LIN {X -0.030,Y -571.399,Z 1067.188,A 0.000,B 0.000,C 90.000,E1 69.752} C_DIS
LIN {X -0.071,Y -572.958,Z 1067.177,A 0.000,B 0.000,C 90.000,E1 67.847} C_DIS
LIN {X -0.064,Y -573.976,Z 1067.169,A 0.000,B 0.000,C 90.000,E1 66.485} C_DIS
LIN {X -0.020,Y -574.631,Z 1067.165,A 0.000,B 0.000,C 90.000,E1 65.665} C_DIS
LIN {X 0.089,Y -575.617,Z 1067.156,A 0.000,B 0.000,C 90.000,E1 64.024} C_DIS
LIN {X -0.046,Y -576.546,Z 1067.147,A 0.000,B 0.000,C 90.000,E1 62.410} C_DIS
LIN {X -0.162,Y -577.447,Z 1067.138,A 0.000,B 0.000,C 90.000,E1 60.795} C_DIS
LIN {X 0.161,Y -578.076,Z 1067.130,A 0.000,B 0.000,C 90.000,E1 59.410} C_DIS
LIN {X 0.146,Y -578.736,Z 1067.121,A 0.000,B 0.000,C 90.000,E1 57.788} C_DIS
LIN {X 0.303,Y -579.331,Z 1067.114,A 0.000,B 0.000,C 90.000,E1 56.421} C_DIS
LIN {X 0.155,Y -579.956,Z 1067.105,A 0.000,B 0.000,C 90.000,E1 54.815} C_DIS
LIN {X 0.019,Y -580.235,Z 1067.099,A 0.000,B 0.000,C 90.000,E1 53.749} C_DIS
LIN {X 0.058,Y -580.388,Z 1067.091,A 0.000,B 0.000,C 90.000,E1 52.396} C_DIS
LIN {X -0.248,Y -580.373,Z 1067.087,A 0.000,B 0.000,C 90.000,E1 51.618} C_DIS
LIN {X -0.198,Y -580.244,Z 1067.082,A 0.000,B 0.000,C 90.000,E1 50.803} C_DIS
LIN {X -0.386,Y -579.481,Z 1067.072,A 0.000,B 0.000,C 90.000,E1 48.933} C_DIS
LIN {X -0.089,Y -578.838,Z 1067.064,A 0.000,B 0.000,C 90.000,E1 47.553} C_DIS
LIN {X 0.044,Y -578.138,Z 1067.058,A 0.000,B 0.000,C 90.000,E1 46.458} C_DIS
LIN {X -0.249,Y -577.299,Z 1067.052,A 0.000,B 0.000,C 90.000,E1 45.405} C_DIS
LIN {X -0.269,Y -576.458,Z 1067.048,A 0.000,B 0.000,C 90.000,E1 44.595} C_DIS
LIN {X 0.229,Y -575.023,Z 1067.042,A 0.000,B 0.000,C 90.000,E1 43.461} C_DIS
LIN {X -0.082,Y -573.483,Z 1067.036,A 0.000,B 0.000,C 90.000,E1 42.405} C_DIS
LIN {X -0.022,Y -571.800,Z 1067.030,A 0.000,B 0.000,C 90.000,E1 41.310} C_DIS
LIN {X -0.191,Y -570.844,Z 1067.026,A 0.000,B 0.000,C 90.000,E1 40.782} C_DIS
LIN {X 0.253,Y -568.409,Z 1067.020,A 0.000,B 0.000,C 90.000,E1 39.644} C_DIS
LIN {X -0.146,Y -565.732,Z 1067.014,A 0.000,B 0.000,C 90.000,E1 38.588} C_DIS
LIN {X 0.192,Y -563.413,Z 1067.010,A 0.000,B 0.000,C 90.000,E1 37.729} C_DIS
LIN {X -0.043,Y -561.737,Z 1067.007,A 0.000,B 0.000,C 90.000,E1 37.202} C_DIS
LIN {X -0.180,Y -559.895,Z 1067.004,A 0.000,B 0.000,C 90.000,E1 36.664} C_DIS
LIN {X 0.010,Y -557.860,Z 1067.001,A 0.000,B 0.000,C 90.000,E1 36.091} C_DIS
LIN {X 0.018,Y -553.342,Z 1066.994,A 0.000,B 0.000,C 90.000,E1 34.978} C_DIS
LIN {X 0.214,Y -549.557,Z 1066.990,A 0.000,B 0.000,C 90.000,E1 34.119} C_DIS
LIN {X -0.080,Y -544.761,Z 1066.984,A 0.000,B 0.000,C 90.000,E1 33.166} C_DIS
LIN {X 0.042,Y -537.992,Z 1066.977,A 0.000,B 0.000,C 90.000,E1 31.878} C_DIS
LIN {X -0.102,Y -533.870,Z 1066.973,A 0.000,B 0.000,C 90.000,E1 31.180} C_DIS
LIN {X 0.045,Y -530.368,Z 1066.970,A 0.000,B 0.000,C 90.000,E1 30.590} C_DIS
LIN {X 0.016,Y -525.637,Z 1066.966,A 0.000,B 0.000,C 90.000,E1 29.873} C_DIS
LIN {X -0.191,Y -522.614,Z 1066.964,A 0.000,B 0.000,C 90.000,E1 29.461} C_DIS
LIN {X 0.000,Y -516.123,Z 1066.959,A 0.000,B 0.000,C 90.000,E1 28.565} C_DIS
LIN {X -0.151,Y -510.113,Z 1066.955,A 0.000,B 0.000,C 90.000,E1 27.847} C_DIS
LIN {X -0.175,Y -505.036,Z 1066.951,A 0.000,B 0.000,C 90.000,E1 27.257} C_DIS
LIN {X -0.003,Y -499.864,Z 1066.948,A 0.000,B 0.000,C 90.000,E1 26.668} C_DIS
LIN {X -0.236,Y -491.728,Z 1066.943,A 0.000,B 0.000,C 90.000,E1 25.848} C_DIS
LIN {X -0.003,Y -483.135,Z 1066.939,A 0.000,B 0.000,C 90.000,E1 24.975} C_DIS
LIN {X -0.157,Y -476.253,Z 1066.935,A 0.000,B 0.000,C 90.000,E1 24.335} C_DIS
LIN {X -0.036,Y -468.892,Z 1066.931,A 0.000,B 0.000,C 90.000,E1 23.643} C_DIS
LIN {X 0.046,Y -458.306,Z 1066.926,A 0.000,B 0.000,C 90.000,E1 22.717} C_DIS
LIN {X -0.028,Y -440.218,Z 1066.918,A 0.000,B 0.000,C 90.000,E1 21.153} C_DIS
LIN {X 0.004,Y -425.575,Z 1066.910,A 0.000,B 0.000,C 90.000,E1 19.758} C_DIS
LIN {X -0.051,Y -412.827,Z 1066.902,A 0.000,B 0.000,C 90.000,E1 18.417} C_DIS
LIN {X 0.169,Y -401.988,Z 1066.895,A 0.000,B 0.000,C 90.000,E1 17.094} C_DIS
LIN {X -0.201,Y -399.427,Z 1066.893,A 0.000,B 0.000,C 90.000,E1 16.804} C_DIS
LIN {X -0.053,Y -396.452,Z 1066.891,A 0.000,B 0.000,C 90.000,E1 16.315} C_DIS
LIN {X -0.057,Y -393.760,Z 1066.888,A 0.000,B 0.000,C 90.000,E1 15.788} C_DIS
LIN {X 0.002,Y -392.685,Z 1066.886,A 0.000,B 0.000,C 90.000,E1 15.426} C_DIS
LIN {X 0.027,Y -392.266,Z 1066.885,A 0.000,B 0.000,C 90.000,E1 15.245} C_DIS
LIN {X -0.004,Y -391.751,Z 1066.882,A 0.000,B 0.000,C 90.000,E1 14.717} C_DIS
LIN {X -0.013,Y -391.981,Z 1066.878,A 0.000,B 0.000,C 90.000,E1 14.008} C_DIS
LIN {X -0.033,Y -394.540,Z 1066.866,A 0.000,B 0.000,C 90.000,E1 11.883} C_DIS
LIN {X 0.072,Y -401.042,Z 1066.844,A 0.000,B 0.000,C 90.000,E1 7.992} C_DIS
LIN {X -0.059,Y -406.203,Z 1066.831,A 0.000,B 0.000,C 90.000,E1 5.568} C_DIS
LIN {X -0.104,Y -409.358,Z 1066.823,A 0.000,B 0.000,C 90.000,E1 4.188} C_DIS
LIN {X -0.094,Y -410.505,Z 1066.821,A 0.000,B 0.000,C 90.000,E1 3.841} C_DIS
LIN {X -0.107,Y -411.862,Z 1066.819,A 0.000,B 0.000,C 90.000,E1 3.498} C_DIS
LIN {X 0.103,Y -416.825,Z 1066.815,A 0.000,B 0.000,C 90.000,E1 2.751} C_DIS
LIN {X -0.106,Y -417.565,Z 1066.815,A 0.000,B 0.000,C 90.000,E1 2.694} C_DIS
LIN {X 0.187,Y -422.034,Z 1066.813,A 0.000,B 0.000,C 90.000,E1 2.293} C_DIS
LIN {X -0.034,Y -437.430,Z 1066.807,A 0.000,B 0.000,C 90.000,E1 1.318} C_DIS
LIN {X 0.000,Y -458.071,Z 1066.800,A 0.000,B 0.000,C 90.000,E1 360.000} C_DIS
LIN {X 0.211,Y -476.247,Z 1066.794,A 0.000,B 0.000,C 90.000,E1 358.854} C_DIS
LIN {X 0.190,Y -489.260,Z 1066.789,A 0.000,B 0.000,C 90.000,E1 358.051} C_DIS
LIN {X -0.172,Y -500.347,Z 1066.785,A 0.000,B 0.000,C 90.000,E1 357.364} C_DIS
LIN {X 0.093,Y -506.513,Z 1066.783,A 0.000,B 0.000,C 90.000,E1 356.906} C_DIS
LIN {X 0.224,Y -511.098,Z 1066.781,A 0.000,B 0.000,C 90.000,E1 356.560} C_DIS
LIN {X 0.246,Y -517.071,Z 1066.779,A 0.000,B 0.000,C 90.000,E1 356.102} C_DIS
LIN {X 0.102,Y -522.907,Z 1066.776,A 0.000,B 0.000,C 90.000,E1 355.641} C_DIS
LIN {X 0.123,Y -529.896,Z 1066.772,A 0.000,B 0.000,C 90.000,E1 355.008} C_DIS
LIN {X -0.052,Y -536.533,Z 1066.769,A 0.000,B 0.000,C 90.000,E1 354.375} C_DIS
LIN {X -0.053,Y -542.882,Z 1066.765,A 0.000,B 0.000,C 90.000,E1 353.685} C_DIS
LIN {X 0.032,Y -547.721,Z 1066.762,A 0.000,B 0.000,C 90.000,E1 353.109} C_DIS
LIN {X -0.031,Y -552.917,Z 1066.758,A 0.000,B 0.000,C 90.000,E1 352.413} C_DIS
LIN {X -0.073,Y -557.579,Z 1066.754,A 0.000,B 0.000,C 90.000,E1 351.724} C_DIS
LIN {X 0.200,Y -560.989,Z 1066.751,A 0.000,B 0.000,C 90.000,E1 351.141} C_DIS
LIN {X 0.260,Y -564.855,Z 1066.747,A 0.000,B 0.000,C 90.000,E1 350.443} C_DIS
LIN {X -0.205,Y -568.367,Z 1066.743,A 0.000,B 0.000,C 90.000,E1 349.803} C_DIS
LIN {X 0.158,Y -570.958,Z 1066.740,A 0.000,B 0.000,C 90.000,E1 349.218} C_DIS
LIN {X 0.065,Y -574.652,Z 1066.736,A 0.000,B 0.000,C 90.000,E1 348.409} C_DIS
LIN {X -0.236,Y -579.214,Z 1066.730,A 0.000,B 0.000,C 90.000,E1 347.353} C_DIS
LIN {X 0.225,Y -583.442,Z 1066.724,A 0.000,B 0.000,C 90.000,E1 346.228} C_DIS
LIN {X -0.202,Y -586.421,Z 1066.719,A 0.000,B 0.000,C 90.000,E1 345.463} C_DIS
LIN {X 0.053,Y -591.220,Z 1066.712,A 0.000,B 0.000,C 90.000,E1 344.102} C_DIS
LIN {X -0.012,Y -595.796,Z 1066.704,A 0.000,B 0.000,C 90.000,E1 342.779} C_DIS
LIN {X 0.005,Y -600.020,Z 1066.697,A 0.000,B 0.000,C 90.000,E1 341.456} C_DIS
LIN {X -0.196,Y -603.025,Z 1066.691,A 0.000,B 0.000,C 90.000,E1 340.423} C_DIS
LIN {X 0.209,Y -605.887,Z 1066.685,A 0.000,B 0.000,C 90.000,E1 339.337} C_DIS
LIN {X 0.016,Y -609.144,Z 1066.678,A 0.000,B 0.000,C 90.000,E1 338.050} C_DIS
LIN {X 0.148,Y -611.467,Z 1066.672,A 0.000,B 0.000,C 90.000,E1 336.997} C_DIS
LIN {X -0.002,Y -613.490,Z 1066.667,A 0.000,B 0.000,C 90.000,E1 335.973} C_DIS
LIN {X 0.188,Y -615.254,Z 1066.661,A 0.000,B 0.000,C 90.000,E1 334.921} C_DIS
LIN {X 0.120,Y -616.362,Z 1066.656,A 0.000,B 0.000,C 90.000,E1 334.152} C_DIS
LIN {X 0.050,Y -617.801,Z 1066.651,A 0.000,B 0.000,C 90.000,E1 333.127} C_DIS
LIN {X -0.014,Y -619.315,Z 1066.644,A 0.000,B 0.000,C 90.000,E1 331.847} C_DIS
LIN {X 0.242,Y -620.351,Z 1066.638,A 0.000,B 0.000,C 90.000,E1 330.795} C_DIS
LIN {X -0.023,Y -621.098,Z 1066.632,A 0.000,B 0.000,C 90.000,E1 329.793} C_DIS
LIN {X 0.259,Y -621.563,Z 1066.626,A 0.000,B 0.000,C 90.000,E1 328.742} C_DIS
LIN {X 0.324,Y -621.879,Z 1066.619,A 0.000,B 0.000,C 90.000,E1 327.454} C_DIS
LIN {X 0.412,Y -621.733,Z 1066.614,A 0.000,B 0.000,C 90.000,E1 326.421} C_DIS
LIN {X 0.284,Y -621.081,Z 1066.605,A 0.000,B 0.000,C 90.000,E1 324.895} C_DIS
LIN {X 0.176,Y -620.378,Z 1066.598,A 0.000,B 0.000,C 90.000,E1 323.623} C_DIS
LIN {X -0.120,Y -619.547,Z 1066.589,A 0.000,B 0.000,C 90.000,E1 322.110} C_DIS
LIN {X -0.304,Y -618.323,Z 1066.574,A 0.000,B 0.000,C 90.000,E1 319.299} C_DIS
LIN {X 0.132,Y -617.702,Z 1066.565,A 0.000,B 0.000,C 90.000,E1 317.715} C_DIS
LIN {X 0.193,Y -616.713,Z 1066.554,A 0.000,B 0.000,C 90.000,E1 315.648} C_DIS
LIN {X 0.112,Y -615.929,Z 1066.545,A 0.000,B 0.000,C 90.000,E1 314.109} C_DIS
LIN {X -0.249,Y -615.415,Z 1066.538,A 0.000,B 0.000,C 90.000,E1 312.852} C_DIS
LIN {X 0.245,Y -614.698,Z 1066.531,A 0.000,B 0.000,C 90.000,E1 311.515} C_DIS
LIN {X -0.037,Y -614.260,Z 1066.528,A 0.000,B 0.000,C 90.000,E1 311.024} C_DIS
LIN {X 0.085,Y -614.051,Z 1066.525,A 0.000,B 0.000,C 90.000,E1 310.496} C_DIS
LIN {X -0.088,Y -613.785,Z 1066.524,A 0.000,B 0.000,C 90.000,E1 310.253} C_DIS
LIN {X 0.030,Y -613.623,Z 1066.521,A 0.000,B 0.000,C 90.000,E1 309.725} C_DIS
LIN {X 0.144,Y -613.301,Z 1066.518,A 0.000,B 0.000,C 90.000,E1 309.197} C_DIS
LIN {X -0.039,Y -613.093,Z 1066.516,A 0.000,B 0.000,C 90.000,E1 308.955} C_DIS
LIN {X 0.253,Y -613.081,Z 1066.515,A 0.000,B 0.000,C 90.000,E1 308.669} C_DIS
LIN {X -0.022,Y -612.710,Z 1066.512,A 0.000,B 0.000,C 90.000,E1 308.177} C_DIS
LIN {X 0.080,Y -612.601,Z 1066.509,A 0.000,B 0.000,C 90.000,E1 307.649} C_DIS
LIN {X -0.101,Y -612.222,Z 1066.504,A 0.000,B 0.000,C 90.000,E1 306.629} C_DIS
LIN {X 0.118,Y -611.806,Z 1066.501,A 0.000,B 0.000,C 90.000,E1 306.091} C_DIS
LIN {X -0.088,Y -611.875,Z 1066.499,A 0.000,B 0.000,C 90.000,E1 305.851} C_DIS
LIN {X 0.142,Y -611.376,Z 1066.492,A 0.000,B 0.000,C 90.000,E1 304.532} C_DIS
LIN {X -0.138,Y -610.995,Z 1066.489,A 0.000,B 0.000,C 90.000,E1 304.040} C_DIS
LIN {X -0.116,Y -611.150,Z 1066.488,A 0.000,B 0.000,C 90.000,E1 303.785} C_DIS
LIN {X -0.173,Y -610.869,Z 1066.482,A 0.000,B 0.000,C 90.000,E1 302.752} C_DIS
LIN {X 0.279,Y -610.513,Z 1066.476,A 0.000,B 0.000,C 90.000,E1 301.671} C_DIS
LIN {X 0.153,Y -609.980,Z 1066.469,A 0.000,B 0.000,C 90.000,E1 300.384} C_DIS
LIN {X 0.230,Y -609.001,Z 1066.462,A 0.000,B 0.000,C 90.000,E1 299.077} C_DIS
LIN {X 0.291,Y -607.446,Z 1066.454,A 0.000,B 0.000,C 90.000,E1 297.769} C_DIS
LIN {X 0.145,Y -605.993,Z 1066.450,A 0.000,B 0.000,C 90.000,E1 297.001} C_DIS
LIN {X -0.070,Y -603.682,Z 1066.444,A 0.000,B 0.000,C 90.000,E1 295.976} C_DIS
LIN {X -0.253,Y -600.971,Z 1066.440,A 0.000,B 0.000,C 90.000,E1 295.207} C_DIS
LIN {X 0.153,Y -598.919,Z 1066.437,A 0.000,B 0.000,C 90.000,E1 294.643} C_DIS
LIN {X -0.003,Y -596.261,Z 1066.434,A 0.000,B 0.000,C 90.000,E1 294.131} C_DIS
LIN {X 0.124,Y -592.950,Z 1066.431,A 0.000,B 0.000,C 90.000,E1 293.590} C_DIS
LIN {X -0.023,Y -589.720,Z 1066.429,A 0.000,B 0.000,C 90.000,E1 293.206} C_DIS
LIN {X -0.164,Y -586.074,Z 1066.427,A 0.000,B 0.000,C 90.000,E1 292.823} C_DIS
LIN {X -0.010,Y -575.693,Z 1066.421,A 0.000,B 0.000,C 90.000,E1 291.770} C_DIS
LIN {X -0.243,Y -571.780,Z 1066.419,A 0.000,B 0.000,C 90.000,E1 291.408} C_DIS
LIN {X -0.202,Y -567.332,Z 1066.417,A 0.000,B 0.000,C 90.000,E1 291.046} C_DIS
LIN {X -0.086,Y -565.547,Z 1066.416,A 0.000,B 0.000,C 90.000,E1 290.918} C_DIS
LIN {X 0.092,Y -558.320,Z 1066.415,A 0.000,B 0.000,C 90.000,E1 290.737} C_DIS
LIN {X 0.007,Y -556.592,Z 1066.415,A 0.000,B 0.000,C 90.000,E1 290.737} C_DIS
LIN {X -0.023,Y -549.863,Z 1066.415,A 0.000,B 0.000,C 90.000,E1 290.737} C_DIS
LIN {X 0.042,Y -546.367,Z 1066.415,A 0.000,B 0.000,C 90.000,E1 290.663} C_DIS
LIN {X 0.000,Y -546.303,Z 1066.415,A 0.000,B 0.000,C 90.000,E1 290.663} C_DIS
LIN {X 0.044,Y -546.261,Z 1066.413,A 0.000,B 0.000,C 90.000,E1 290.355} C_DIS
LIN {X 0.107,Y -545.295,Z 1066.412,A 0.000,B 0.000,C 90.000,E1 290.066} C_DIS
LIN {X -0.191,Y -544.391,Z 1066.411,A 0.000,B 0.000,C 90.000,E1 289.939} C_DIS
LIN {X 0.087,Y -544.009,Z 1066.408,A 0.000,B 0.000,C 90.000,E1 289.504} C_DIS
LIN {X 0.182,Y -543.929,Z 1066.396,A 0.000,B 0.000,C 90.000,E1 287.330} C_DIS
LIN {X -0.176,Y -543.745,Z 1066.389,A 0.000,B 0.000,C 90.000,E1 285.953} C_DIS
LIN {X 0.285,Y -543.461,Z 1066.382,A 0.000,B 0.000,C 90.000,E1 284.773} C_DIS
LIN {X -0.145,Y -542.922,Z 1066.373,A 0.000,B 0.000,C 90.000,E1 283.119} C_DIS
LIN {X -0.177,Y -542.028,Z 1066.363,A 0.000,B 0.000,C 90.000,E1 281.422} C_DIS
LIN {X -0.233,Y -541.045,Z 1066.354,A 0.000,B 0.000,C 90.000,E1 279.726} C_DIS
LIN {X 0.047,Y -540.289,Z 1066.346,A 0.000,B 0.000,C 90.000,E1 278.276} C_DIS
LIN {X 0.239,Y -539.273,Z 1066.337,A 0.000,B 0.000,C 90.000,E1 276.549} C_DIS
LIN {X -0.114,Y -538.318,Z 1066.327,A 0.000,B 0.000,C 90.000,E1 274.878} C_DIS
LIN {X 0.040,Y -537.272,Z 1066.316,A 0.000,B 0.000,C 90.000,E1 272.865} C_DIS
LIN {X 0.099,Y -536.330,Z 1066.307,A 0.000,B 0.000,C 90.000,E1 271.146} C_DIS
LIN {X 0.130,Y -535.185,Z 1066.295,A 0.000,B 0.000,C 90.000,E1 269.141} C_DIS
LIN {X 0.145,Y -534.137,Z 1066.286,A 0.000,B 0.000,C 90.000,E1 267.421} C_DIS
LIN {X 0.138,Y -533.253,Z 1066.278,A 0.000,B 0.000,C 90.000,E1 265.988} C_DIS
LIN {X 0.176,Y -532.037,Z 1066.268,A 0.000,B 0.000,C 90.000,E1 264.261} C_DIS
LIN {X 0.188,Y -531.035,Z 1066.262,A 0.000,B 0.000,C 90.000,E1 263.109} C_DIS
LIN {X 0.250,Y -529.841,Z 1066.255,A 0.000,B 0.000,C 90.000,E1 261.951} C_DIS
LIN {X -0.223,Y -527.655,Z 1066.244,A 0.000,B 0.000,C 90.000,E1 259.982} C_DIS
LIN {X -0.096,Y -526.087,Z 1066.236,A 0.000,B 0.000,C 90.000,E1 258.522} C_DIS
LIN {X 0.002,Y -524.587,Z 1066.228,A 0.000,B 0.000,C 90.000,E1 257.061} C_DIS
LIN {X -0.187,Y -522.755,Z 1066.219,A 0.000,B 0.000,C 90.000,E1 255.338} C_DIS
LIN {X -0.042,Y -521.261,Z 1066.210,A 0.000,B 0.000,C 90.000,E1 253.866} C_DIS
LIN {X -0.138,Y -519.757,Z 1066.202,A 0.000,B 0.000,C 90.000,E1 252.417} C_DIS
LIN {X 0.239,Y -518.114,Z 1066.194,A 0.000,B 0.000,C 90.000,E1 250.913} C_DIS
LIN {X 0.129,Y -516.767,Z 1066.188,A 0.000,B 0.000,C 90.000,E1 249.752} C_DIS
LIN {X -0.001,Y -515.383,Z 1066.181,A 0.000,B 0.000,C 90.000,E1 248.592} C_DIS
LIN {X 0.285,Y -512.923,Z 1066.171,A 0.000,B 0.000,C 90.000,E1 246.794} C_DIS
LIN {X -0.181,Y -511.207,Z 1066.165,A 0.000,B 0.000,C 90.000,E1 245.665} C_DIS
LIN {X 0.006,Y -509.401,Z 1066.158,A 0.000,B 0.000,C 90.000,E1 244.460} C_DIS
LIN {X 0.163,Y -507.489,Z 1066.152,A 0.000,B 0.000,C 90.000,E1 243.256} C_DIS
LIN {X -0.166,Y -505.502,Z 1066.145,A 0.000,B 0.000,C 90.000,E1 242.103} C_DIS
LIN {X 0.022,Y -503.021,Z 1066.137,A 0.000,B 0.000,C 90.000,E1 240.589} C_DIS
LIN {X 0.161,Y -500.314,Z 1066.128,A 0.000,B 0.000,C 90.000,E1 239.076} C_DIS
LIN {X -0.057,Y -497.007,Z 1066.118,A 0.000,B 0.000,C 90.000,E1 237.296} C_DIS
LIN {X -0.055,Y -494.697,Z 1066.112,A 0.000,B 0.000,C 90.000,E1 236.087} C_DIS
LIN {X 0.029,Y -491.763,Z 1066.103,A 0.000,B 0.000,C 90.000,E1 234.562} C_DIS
LIN {X -0.056,Y -488.521,Z 1066.095,A 0.000,B 0.000,C 90.000,E1 233.050} C_DIS
LIN {X 0.134,Y -483.667,Z 1066.083,A 0.000,B 0.000,C 90.000,E1 230.884} C_DIS
LIN {X 0.019,Y -480.922,Z 1066.076,A 0.000,B 0.000,C 90.000,E1 229.666} C_DIS
LIN {X 0.244,Y -476.342,Z 1066.064,A 0.000,B 0.000,C 90.000,E1 227.472} C_DIS
LIN {X -0.035,Y -472.065,Z 1066.052,A 0.000,B 0.000,C 90.000,E1 225.324} C_DIS
LIN {X -0.096,Y -467.954,Z 1066.040,A 0.000,B 0.000,C 90.000,E1 223.137} C_DIS
LIN {X 0.215,Y -465.539,Z 1066.033,A 0.000,B 0.000,C 90.000,E1 221.838} C_DIS
LIN {X -0.014,Y -461.635,Z 1066.022,A 0.000,B 0.000,C 90.000,E1 219.967} C_DIS
LIN {X -0.066,Y -458.424,Z 1066.013,A 0.000,B 0.000,C 90.000,E1 218.382} C_DIS
LIN {X -0.021,Y -454.596,Z 1066.003,A 0.000,B 0.000,C 90.000,E1 216.457} C_DIS
LIN {X 0.219,Y -451.201,Z 1065.994,A 0.000,B 0.000,C 90.000,E1 214.818} C_DIS
LIN {X 0.269,Y -446.523,Z 1065.981,A 0.000,B 0.000,C 90.000,E1 212.546} C_DIS
LIN {X 0.214,Y -443.332,Z 1065.972,A 0.000,B 0.000,C 90.000,E1 210.924} C_DIS
LIN {X -0.130,Y -440.084,Z 1065.963,A 0.000,B 0.000,C 90.000,E1 209.333} C_DIS
LIN {X -0.081,Y -434.277,Z 1065.946,A 0.000,B 0.000,C 90.000,E1 206.360} C_DIS
LIN {X -0.039,Y -431.194,Z 1065.937,A 0.000,B 0.000,C 90.000,E1 204.695} C_DIS
LIN {X -0.121,Y -424.184,Z 1065.913,A 0.000,B 0.000,C 90.000,E1 200.355} C_DIS
LIN {X 0.224,Y -422.784,Z 1065.906,A 0.000,B 0.000,C 90.000,E1 198.960} C_DIS
LIN {X 0.015,Y -421.934,Z 1065.898,A 0.000,B 0.000,C 90.000,E1 197.638} C_DIS
LIN {X -0.156,Y -421.916,Z 1065.894,A 0.000,B 0.000,C 90.000,E1 196.985} C_DIS
LIN {X -0.030,Y -422.667,Z 1065.889,A 0.000,B 0.000,C 90.000,E1 195.953} C_DIS
LIN {X 0.211,Y -423.519,Z 1065.885,A 0.000,B 0.000,C 90.000,E1 195.245} C_DIS
LIN {X 0.074,Y -424.984,Z 1065.881,A 0.000,B 0.000,C 90.000,E1 194.592} C_DIS
LIN {X -0.086,Y -427.529,Z 1065.876,A 0.000,B 0.000,C 90.000,E1 193.772} C_DIS
LIN {X -0.114,Y -431.622,Z 1065.871,A 0.000,B 0.000,C 90.000,E1 192.771} C_DIS
LIN {X -0.092,Y -436.531,Z 1065.865,A 0.000,B 0.000,C 90.000,E1 191.771} C_DIS
LIN {X -0.107,Y -451.532,Z 1065.851,A 0.000,B 0.000,C 90.000,E1 189.151} C_DIS
LIN {X -0.083,Y -460.455,Z 1065.843,A 0.000,B 0.000,C 90.000,E1 187.701} C_DIS
LIN {X 0.146,Y -470.184,Z 1065.834,A 0.000,B 0.000,C 90.000,E1 186.087} C_DIS
LIN {X -0.211,Y -477.489,Z 1065.827,A 0.000,B 0.000,C 90.000,E1 184.878} C_DIS
LIN {X 0.164,Y -485.436,Z 1065.819,A 0.000,B 0.000,C 90.000,E1 183.440} C_DIS
LIN {X 0.164,Y -493.274,Z 1065.812,A 0.000,B 0.000,C 90.000,E1 182.064} C_DIS
LIN {X -0.205,Y -500.758,Z 1065.804,A 0.000,B 0.000,C 90.000,E1 180.745} C_DIS
LIN {X 0.140,Y -506.554,Z 1065.798,A 0.000,B 0.000,C 90.000,E1 179.656} C_DIS
LIN {X -0.090,Y -515.402,Z 1065.789,A 0.000,B 0.000,C 90.000,E1 178.051} C_DIS
LIN {X 0.223,Y -520.106,Z 1065.784,A 0.000,B 0.000,C 90.000,E1 177.135} C_DIS
LIN {X -0.238,Y -528.669,Z 1065.775,A 0.000,B 0.000,C 90.000,E1 175.584} C_DIS
LIN {X 0.008,Y -535.597,Z 1065.768,A 0.000,B 0.000,C 90.000,E1 174.261} C_DIS
LIN {X 0.172,Y -544.722,Z 1065.759,A 0.000,B 0.000,C 90.000,E1 172.534} C_DIS
LIN {X 0.026,Y -552.047,Z 1065.751,A 0.000,B 0.000,C 90.000,E1 171.141} C_DIS
LIN {X 0.268,Y -558.542,Z 1065.744,A 0.000,B 0.000,C 90.000,E1 169.859} C_DIS
LIN {X 0.071,Y -564.889,Z 1065.737,A 0.000,B 0.000,C 90.000,E1 168.634} C_DIS
LIN {X -0.159,Y -571.624,Z 1065.729,A 0.000,B 0.000,C 90.000,E1 167.285} C_DIS
LIN {X -0.282,Y -577.965,Z 1065.722,A 0.000,B 0.000,C 90.000,E1 165.936} C_DIS
LIN {X 0.310,Y -584.597,Z 1065.714,A 0.000,B 0.000,C 90.000,E1 164.393} C_DIS
LIN {X 0.294,Y -589.217,Z 1065.708,A 0.000,B 0.000,C 90.000,E1 163.323} C_DIS
LIN {X -0.236,Y -593.466,Z 1065.702,A 0.000,B 0.000,C 90.000,E1 162.308} C_DIS
LIN {X 0.036,Y -597.534,Z 1065.696,A 0.000,B 0.000,C 90.000,E1 161.221} C_DIS
LIN {X 0.276,Y -602.275,Z 1065.688,A 0.000,B 0.000,C 90.000,E1 159.880} C_DIS
LIN {X 0.101,Y -605.753,Z 1065.683,A 0.000,B 0.000,C 90.000,E1 158.847} C_DIS
LIN {X 0.191,Y -609.087,Z 1065.677,A 0.000,B 0.000,C 90.000,E1 157.794} C_DIS
LIN {X 0.289,Y -612.984,Z 1065.670,A 0.000,B 0.000,C 90.000,E1 156.485} C_DIS
LIN {X -0.085,Y -615.960,Z 1065.664,A 0.000,B 0.000,C 90.000,E1 155.485} C_DIS
LIN {X -0.162,Y -618.773,Z 1065.658,A 0.000,B 0.000,C 90.000,E1 154.460} C_DIS
LIN {X -0.194,Y -623.308,Z 1065.648,A 0.000,B 0.000,C 90.000,E1 152.666} C_DIS
LIN {X -0.179,Y -625.209,Z 1065.644,A 0.000,B 0.000,C 90.000,E1 151.897} C_DIS
LIN {X 0.184,Y -628.261,Z 1065.637,A 0.000,B 0.000,C 90.000,E1 150.589} C_DIS
LIN {X 0.030,Y -630.618,Z 1065.631,A 0.000,B 0.000,C 90.000,E1 149.587} C_DIS
LIN {X -0.039,Y -634.001,Z 1065.623,A 0.000,B 0.000,C 90.000,E1 148.074} C_DIS
LIN {X -0.289,Y -636.738,Z 1065.616,A 0.000,B 0.000,C 90.000,E1 146.834} C_DIS
LIN {X -0.095,Y -639.882,Z 1065.607,A 0.000,B 0.000,C 90.000,E1 145.308} C_DIS
LIN {X 0.156,Y -642.978,Z 1065.599,A 0.000,B 0.000,C 90.000,E1 143.783} C_DIS
LIN {X 0.002,Y -645.021,Z 1065.593,A 0.000,B 0.000,C 90.000,E1 142.798} C_DIS
LIN {X -0.246,Y -647.106,Z 1065.588,A 0.000,B 0.000,C 90.000,E1 141.823} C_DIS
LIN {X -0.132,Y -651.192,Z 1065.577,A 0.000,B 0.000,C 90.000,E1 139.828} C_DIS
LIN {X 0.154,Y -653.766,Z 1065.570,A 0.000,B 0.000,C 90.000,E1 138.566} C_DIS
LIN {X 0.426,Y -656.456,Z 1065.563,A 0.000,B 0.000,C 90.000,E1 137.310} C_DIS
LIN {X -0.252,Y -660.903,Z 1065.552,A 0.000,B 0.000,C 90.000,E1 135.405} C_DIS
LIN {X 0.119,Y -667.125,Z 1065.539,A 0.000,B 0.000,C 90.000,E1 132.933} C_DIS
LIN {X -0.327,Y -669.721,Z 1065.533,A 0.000,B 0.000,C 90.000,E1 132.000} C_DIS
LIN {X -0.096,Y -675.450,Z 1065.521,A 0.000,B 0.000,C 90.000,E1 129.806} C_DIS
LIN {X 0.085,Y -678.489,Z 1065.515,A 0.000,B 0.000,C 90.000,E1 128.588} C_DIS
LIN {X -0.363,Y -682.855,Z 1065.505,A 0.000,B 0.000,C 90.000,E1 126.950} C_DIS
LIN {X 0.042,Y -685.951,Z 1065.499,A 0.000,B 0.000,C 90.000,E1 125.724} C_DIS
LIN {X -0.276,Y -689.405,Z 1065.491,A 0.000,B 0.000,C 90.000,E1 124.326} C_DIS
LIN {X -0.199,Y -691.718,Z 1065.485,A 0.000,B 0.000,C 90.000,E1 123.372} C_DIS
LIN {X -0.441,Y -694.570,Z 1065.479,A 0.000,B 0.000,C 90.000,E1 122.212} C_DIS
LIN {X -0.397,Y -697.762,Z 1065.471,A 0.000,B 0.000,C 90.000,E1 120.797} C_DIS
LIN {X -0.229,Y -699.300,Z 1065.467,A 0.000,B 0.000,C 90.000,E1 120.079} C_DIS
LIN {X 0.304,Y -700.484,Z 1065.463,A 0.000,B 0.000,C 90.000,E1 119.333} C_DIS
LIN {X -0.115,Y -701.345,Z 1065.459,A 0.000,B 0.000,C 90.000,E1 118.665} C_DIS
LIN {X 0.151,Y -703.547,Z 1065.446,A 0.000,B 0.000,C 90.000,E1 116.309} C_DIS
LIN {X 0.372,Y -704.242,Z 1065.442,A 0.000,B 0.000,C 90.000,E1 115.591} C_DIS
LIN {X -0.064,Y -704.784,Z 1065.437,A 0.000,B 0.000,C 90.000,E1 114.695} C_DIS
LIN {X 0.216,Y -704.477,Z 1065.435,A 0.000,B 0.000,C 90.000,E1 114.207} C_DIS
LIN {X -0.143,Y -704.217,Z 1065.433,A 0.000,B 0.000,C 90.000,E1 114.003} C_DIS
LIN {X 0.137,Y -702.824,Z 1065.431,A 0.000,B 0.000,C 90.000,E1 113.515} C_DIS
LIN {X 0.137,Y -701.859,Z 1065.429,A 0.000,B 0.000,C 90.000,E1 113.281} C_DIS
LIN {X 0.037,Y -698.461,Z 1065.427,A 0.000,B 0.000,C 90.000,E1 112.823} C_DIS
LIN {X -0.102,Y -697.441,Z 1065.426,A 0.000,B 0.000,C 90.000,E1 112.717} C_DIS
LIN {X 0.028,Y -695.908,Z 1065.426,A 0.000,B 0.000,C 90.000,E1 112.589} C_DIS
LIN {X 0.391,Y -688.344,Z 1065.424,A 0.000,B 0.000,C 90.000,E1 112.206} C_DIS
LIN {X 0.140,Y -686.479,Z 1065.423,A 0.000,B 0.000,C 90.000,E1 112.153} C_DIS
LIN {X 0.148,Y -683.341,Z 1065.423,A 0.000,B 0.000,C 90.000,E1 112.078} C_DIS
LIN {X -0.276,Y -676.246,Z 1065.422,A 0.000,B 0.000,C 90.000,E1 112.025} C_DIS
LIN {X -0.336,Y -670.336,Z 1065.422,A 0.000,B 0.000,C 90.000,E1 112.025} C_DIS
LIN {X 0.210,Y -608.226,Z 1065.422,A 0.000,B 0.000,C 90.000,E1 111.972} C_DIS
LIN {X -0.063,Y -604.126,Z 1065.421,A 0.000,B 0.000,C 90.000,E1 111.844} C_DIS
LIN {X -0.017,Y -602.506,Z 1065.421,A 0.000,B 0.000,C 90.000,E1 111.770} C_DIS
LIN {X 0.076,Y -596.370,Z 1065.419,A 0.000,B 0.000,C 90.000,E1 111.408} C_DIS
LIN {X 0.036,Y -590.498,Z 1065.417,A 0.000,B 0.000,C 90.000,E1 110.972} C_DIS
LIN {X 0.025,Y -579.590,Z 1065.411,A 0.000,B 0.000,C 90.000,E1 110.066} C_DIS
LIN {X 0.148,Y -575.310,Z 1065.410,A 0.000,B 0.000,C 90.000,E1 109.704} C_DIS
LIN {X -0.020,Y -569.264,Z 1065.407,A 0.000,B 0.000,C 90.000,E1 109.268} C_DIS
LIN {X -0.216,Y -560.881,Z 1065.404,A 0.000,B 0.000,C 90.000,E1 108.779} C_DIS
LIN {X -0.243,Y -554.371,Z 1065.402,A 0.000,B 0.000,C 90.000,E1 108.417} C_DIS
LIN {X -0.083,Y -549.269,Z 1065.400,A 0.000,B 0.000,C 90.000,E1 108.055} C_DIS
LIN {X -0.175,Y -547.691,Z 1065.399,A 0.000,B 0.000,C 90.000,E1 107.873} C_DIS
LIN {X -0.214,Y -547.668,Z 1065.399,A 0.000,B 0.000,C 90.000,E1 107.873} C_DIS
LIN {X -0.042,Y -547.371,Z 1065.398,A 0.000,B 0.000,C 90.000,E1 107.638} C_DIS
LIN {X -0.231,Y -547.440,Z 1065.395,A 0.000,B 0.000,C 90.000,E1 107.094} C_DIS
LIN {X 0.101,Y -548.499,Z 1065.385,A 0.000,B 0.000,C 90.000,E1 105.371} C_DIS
LIN {X 0.243,Y -550.326,Z 1065.371,A 0.000,B 0.000,C 90.000,E1 102.827} C_DIS
LIN {X -0.039,Y -552.057,Z 1065.361,A 0.000,B 0.000,C 90.000,E1 100.894} C_DIS
LIN {X 0.281,Y -554.447,Z 1065.348,A 0.000,B 0.000,C 90.000,E1 98.624} C_DIS
LIN {X -0.232,Y -556.373,Z 1065.339,A 0.000,B 0.000,C 90.000,E1 97.004} C_DIS
LIN {X 0.140,Y -557.656,Z 1065.333,A 0.000,B 0.000,C 90.000,E1 95.853} C_DIS
LIN {X 0.054,Y -558.939,Z 1065.325,A 0.000,B 0.000,C 90.000,E1 94.473} C_DIS
LIN {X -0.134,Y -559.698,Z 1065.319,A 0.000,B 0.000,C 90.000,E1 93.383} C_DIS
LIN {X -0.105,Y -560.546,Z 1065.310,A 0.000,B 0.000,C 90.000,E1 91.718} C_DIS
LIN {X -0.193,Y -561.149,Z 1065.302,A 0.000,B 0.000,C 90.000,E1 90.344} C_DIS
LIN {X -0.169,Y -561.765,Z 1065.293,A 0.000,B 0.000,C 90.000,E1 88.682} C_DIS
LIN {X 0.100,Y -562.588,Z 1065.280,A 0.000,B 0.000,C 90.000,E1 86.445} C_DIS
LIN {X 0.196,Y -563.191,Z 1065.271,A 0.000,B 0.000,C 90.000,E1 84.780} C_DIS
LIN {X 0.263,Y -563.559,Z 1065.264,A 0.000,B 0.000,C 90.000,E1 83.394} C_DIS
LIN {X 0.022,Y -564.120,Z 1065.253,A 0.000,B 0.000,C 90.000,E1 81.489} C_DIS
LIN {X 0.029,Y -564.919,Z 1065.241,A 0.000,B 0.000,C 90.000,E1 79.285} C_DIS
LIN {X -0.290,Y -565.972,Z 1065.228,A 0.000,B 0.000,C 90.000,E1 77.117} C_DIS
LIN {X -0.071,Y -567.082,Z 1065.218,A 0.000,B 0.000,C 90.000,E1 75.172} C_DIS
LIN {X 0.103,Y -568.699,Z 1065.205,A 0.000,B 0.000,C 90.000,E1 72.960} C_DIS
LIN {X 0.153,Y -570.214,Z 1065.195,A 0.000,B 0.000,C 90.000,E1 71.040} C_DIS
LIN {X -0.097,Y -571.394,Z 1065.187,A 0.000,B 0.000,C 90.000,E1 69.699} C_DIS
LIN {X -0.145,Y -572.952,Z 1065.177,A 0.000,B 0.000,C 90.000,E1 67.794} C_DIS
LIN {X 0.086,Y -573.949,Z 1065.169,A 0.000,B 0.000,C 90.000,E1 66.410} C_DIS
LIN {X -0.104,Y -574.561,Z 1065.165,A 0.000,B 0.000,C 90.000,E1 65.613} C_DIS
LIN {X 0.097,Y -575.719,Z 1065.154,A 0.000,B 0.000,C 90.000,E1 63.691} C_DIS
LIN {X -0.297,Y -576.575,Z 1065.145,A 0.000,B 0.000,C 90.000,E1 62.103} C_DIS
LIN {X -0.121,Y -577.227,Z 1065.139,A 0.000,B 0.000,C 90.000,E1 61.001} C_DIS
LIN {X 0.194,Y -577.881,Z 1065.131,A 0.000,B 0.000,C 90.000,E1 59.616} C_DIS
LIN {X 0.171,Y -578.509,Z 1065.122,A 0.000,B 0.000,C 90.000,E1 57.995} C_DIS
LIN {X 0.323,Y -579.078,Z 1065.115,A 0.000,B 0.000,C 90.000,E1 56.628} C_DIS
LIN {X -0.321,Y -579.424,Z 1065.110,A 0.000,B 0.000,C 90.000,E1 55.881} C_DIS
LIN {X 0.334,Y -579.938,Z 1065.101,A 0.000,B 0.000,C 90.000,E1 54.196} C_DIS
LIN {X 0.195,Y -580.123,Z 1065.095,A 0.000,B 0.000,C 90.000,E1 53.130} C_DIS
LIN {X -0.236,Y -580.180,Z 1065.088,A 0.000,B 0.000,C 90.000,E1 51.823} C_DIS
LIN {X -0.019,Y -579.975,Z 1065.082,A 0.000,B 0.000,C 90.000,E1 50.723} C_DIS
LIN {X 0.069,Y -579.329,Z 1065.073,A 0.000,B 0.000,C 90.000,E1 49.094} C_DIS
LIN {X 0.207,Y -578.843,Z 1065.067,A 0.000,B 0.000,C 90.000,E1 48.000} C_DIS
LIN {X 0.069,Y -578.005,Z 1065.059,A 0.000,B 0.000,C 90.000,E1 46.662} C_DIS
LIN {X 0.193,Y -577.157,Z 1065.053,A 0.000,B 0.000,C 90.000,E1 45.567} C_DIS
LIN {X -0.111,Y -576.034,Z 1065.047,A 0.000,B 0.000,C 90.000,E1 44.514} C_DIS
LIN {X 0.091,Y -574.210,Z 1065.040,A 0.000,B 0.000,C 90.000,E1 43.137} C_DIS
LIN {X -0.229,Y -572.569,Z 1065.034,A 0.000,B 0.000,C 90.000,E1 42.081} C_DIS
LIN {X 0.115,Y -571.255,Z 1065.029,A 0.000,B 0.000,C 90.000,E1 41.229} C_DIS
LIN {X -0.058,Y -570.254,Z 1065.026,A 0.000,B 0.000,C 90.000,E1 40.701} C_DIS
LIN {X 0.013,Y -567.801,Z 1065.020,A 0.000,B 0.000,C 90.000,E1 39.600} C_DIS
LIN {X 0.292,Y -565.782,Z 1065.016,A 0.000,B 0.000,C 90.000,E1 38.749} C_DIS
LIN {X 0.185,Y -563.470,Z 1065.011,A 0.000,B 0.000,C 90.000,E1 37.935} C_DIS
LIN {X 0.056,Y -561.839,Z 1065.008,A 0.000,B 0.000,C 90.000,E1 37.397} C_DIS
LIN {X -0.090,Y -559.020,Z 1065.003,A 0.000,B 0.000,C 90.000,E1 36.583} C_DIS
LIN {X 0.091,Y -556.939,Z 1065.000,A 0.000,B 0.000,C 90.000,E1 36.011} C_DIS
LIN {X -0.041,Y -551.721,Z 1064.993,A 0.000,B 0.000,C 90.000,E1 34.771} C_DIS
LIN {X 0.133,Y -547.814,Z 1064.989,A 0.000,B 0.000,C 90.000,E1 33.913} C_DIS
LIN {X -0.180,Y -542.892,Z 1064.983,A 0.000,B 0.000,C 90.000,E1 32.959} C_DIS
LIN {X 0.053,Y -536.740,Z 1064.977,A 0.000,B 0.000,C 90.000,E1 31.799} C_DIS
LIN {X 0.205,Y -531.705,Z 1064.972,A 0.000,B 0.000,C 90.000,E1 30.924} C_DIS
LIN {X 0.185,Y -527.117,Z 1064.968,A 0.000,B 0.000,C 90.000,E1 30.207} C_DIS
LIN {X -0.170,Y -523.226,Z 1064.965,A 0.000,B 0.000,C 90.000,E1 29.667} C_DIS
LIN {X -0.259,Y -517.850,Z 1064.961,A 0.000,B 0.000,C 90.000,E1 28.949} C_DIS
LIN {X -0.056,Y -514.498,Z 1064.958,A 0.000,B 0.000,C 90.000,E1 28.487} C_DIS
LIN {X 0.047,Y -507.157,Z 1064.953,A 0.000,B 0.000,C 90.000,E1 27.590} C_DIS
LIN {X -0.124,Y -500.617,Z 1064.949,A 0.000,B 0.000,C 90.000,E1 26.873} C_DIS
LIN {X 0.101,Y -491.027,Z 1064.944,A 0.000,B 0.000,C 90.000,E1 25.848} C_DIS
LIN {X 0.093,Y -480.038,Z 1064.938,A 0.000,B 0.000,C 90.000,E1 24.771} C_DIS
LIN {X -0.266,Y -470.218,Z 1064.933,A 0.000,B 0.000,C 90.000,E1 23.898} C_DIS
LIN {X -0.031,Y -461.142,Z 1064.928,A 0.000,B 0.000,C 90.000,E1 23.078} C_DIS
LIN {X 0.097,Y -447.536,Z 1064.922,A 0.000,B 0.000,C 90.000,E1 21.897} C_DIS
LIN {X -0.148,Y -429.718,Z 1064.913,A 0.000,B 0.000,C 90.000,E1 20.301} C_DIS
LIN {X 0.176,Y -415.317,Z 1064.905,A 0.000,B 0.000,C 90.000,E1 18.779} C_DIS
LIN {X 0.067,Y -404.233,Z 1064.897,A 0.000,B 0.000,C 90.000,E1 17.511} C_DIS
LIN {X -0.185,Y -400.210,Z 1064.895,A 0.000,B 0.000,C 90.000,E1 17.040} C_DIS
LIN {X -0.019,Y -395.735,Z 1064.891,A 0.000,B 0.000,C 90.000,E1 16.315} C_DIS
LIN {X -0.083,Y -393.559,Z 1064.888,A 0.000,B 0.000,C 90.000,E1 15.898} C_DIS
LIN {X 0.069,Y -392.249,Z 1064.886,A 0.000,B 0.000,C 90.000,E1 15.426} C_DIS
LIN {X -0.089,Y -391.707,Z 1064.882,A 0.000,B 0.000,C 90.000,E1 14.828} C_DIS
LIN {X -0.102,Y -391.981,Z 1064.878,A 0.000,B 0.000,C 90.000,E1 14.120} C_DIS
LIN {X -0.115,Y -392.702,Z 1064.875,A 0.000,B 0.000,C 90.000,E1 13.411} C_DIS
LIN {X 0.035,Y -398.400,Z 1064.853,A 0.000,B 0.000,C 90.000,E1 9.500} C_DIS
LIN {X -0.123,Y -403.020,Z 1064.839,A 0.000,B 0.000,C 90.000,E1 7.068} C_DIS
LIN {X 0.178,Y -409.184,Z 1064.824,A 0.000,B 0.000,C 90.000,E1 4.245} C_DIS
LIN {X 0.188,Y -410.153,Z 1064.822,A 0.000,B 0.000,C 90.000,E1 3.898} C_DIS
LIN {X 0.173,Y -411.313,Z 1064.820,A 0.000,B 0.000,C 90.000,E1 3.555} C_DIS
LIN {X 0.169,Y -412.154,Z 1064.819,A 0.000,B 0.000,C 90.000,E1 3.383} C_DIS
LIN {X 0.080,Y -416.988,Z 1064.815,A 0.000,B 0.000,C 90.000,E1 2.694} C_DIS
LIN {X -0.014,Y -419.045,Z 1064.814,A 0.000,B 0.000,C 90.000,E1 2.522} C_DIS
LIN {X -0.214,Y -422.057,Z 1064.813,A 0.000,B 0.000,C 90.000,E1 2.293} C_DIS
LIN {X -0.101,Y -437.634,Z 1064.807,A 0.000,B 0.000,C 90.000,E1 1.260} C_DIS
LIN {X 0.000,Y -457.259,Z 1064.800,A 0.000,B 0.000,C 90.000,E1 360.000} C_DIS
LIN {X 0.080,Y -473.783,Z 1064.794,A 0.000,B 0.000,C 90.000,E1 358.969} C_DIS
LIN {X 0.117,Y -486.793,Z 1064.790,A 0.000,B 0.000,C 90.000,E1 358.165} C_DIS
LIN {X 0.237,Y -496.420,Z 1064.786,A 0.000,B 0.000,C 90.000,E1 357.535} C_DIS
LIN {X 0.180,Y -504.161,Z 1064.784,A 0.000,B 0.000,C 90.000,E1 357.020} C_DIS
LIN {X -0.069,Y -511.722,Z 1064.781,A 0.000,B 0.000,C 90.000,E1 356.502} C_DIS
LIN {X -0.109,Y -517.709,Z 1064.778,A 0.000,B 0.000,C 90.000,E1 356.045} C_DIS
LIN {X -0.193,Y -523.459,Z 1064.775,A 0.000,B 0.000,C 90.000,E1 355.584} C_DIS
LIN {X -0.142,Y -530.413,Z 1064.772,A 0.000,B 0.000,C 90.000,E1 354.951} C_DIS
LIN {X -0.020,Y -536.732,Z 1064.768,A 0.000,B 0.000,C 90.000,E1 354.318} C_DIS
LIN {X -0.020,Y -543.090,Z 1064.765,A 0.000,B 0.000,C 90.000,E1 353.628} C_DIS
LIN {X 0.215,Y -547.795,Z 1064.762,A 0.000,B 0.000,C 90.000,E1 353.053} C_DIS
LIN {X 0.261,Y -552.949,Z 1064.758,A 0.000,B 0.000,C 90.000,E1 352.356} C_DIS
LIN {X -0.079,Y -556.764,Z 1064.755,A 0.000,B 0.000,C 90.000,E1 351.837} C_DIS
LIN {X -0.060,Y -561.076,Z 1064.751,A 0.000,B 0.000,C 90.000,E1 351.141} C_DIS
LIN {X 0.152,Y -564.251,Z 1064.748,A 0.000,B 0.000,C 90.000,E1 350.566} C_DIS
LIN {X 0.094,Y -568.540,Z 1064.743,A 0.000,B 0.000,C 90.000,E1 349.746} C_DIS
LIN {X -0.103,Y -571.145,Z 1064.740,A 0.000,B 0.000,C 90.000,E1 349.218} C_DIS
LIN {X 0.244,Y -575.469,Z 1064.735,A 0.000,B 0.000,C 90.000,E1 348.229} C_DIS
LIN {X -0.040,Y -580.011,Z 1064.729,A 0.000,B 0.000,C 90.000,E1 347.173} C_DIS
LIN {X -0.270,Y -584.229,Z 1064.723,A 0.000,B 0.000,C 90.000,E1 346.117} C_DIS
LIN {X 0.194,Y -590.103,Z 1064.714,A 0.000,B 0.000,C 90.000,E1 344.464} C_DIS
LIN {X -0.017,Y -592.934,Z 1064.709,A 0.000,B 0.000,C 90.000,E1 343.685} C_DIS
LIN {X 0.246,Y -596.628,Z 1064.703,A 0.000,B 0.000,C 90.000,E1 342.598} C_DIS
LIN {X 0.279,Y -600.814,Z 1064.696,A 0.000,B 0.000,C 90.000,E1 341.275} C_DIS
LIN {X 0.090,Y -603.810,Z 1064.690,A 0.000,B 0.000,C 90.000,E1 340.242} C_DIS
LIN {X -0.062,Y -606.636,Z 1064.685,A 0.000,B 0.000,C 90.000,E1 339.209} C_DIS
LIN {X -0.241,Y -609.884,Z 1064.677,A 0.000,B 0.000,C 90.000,E1 337.922} C_DIS
LIN {X -0.098,Y -612.213,Z 1064.672,A 0.000,B 0.000,C 90.000,E1 336.869} C_DIS
LIN {X 0.324,Y -614.232,Z 1064.666,A 0.000,B 0.000,C 90.000,E1 335.793} C_DIS
LIN {X -0.037,Y -615.994,Z 1064.660,A 0.000,B 0.000,C 90.000,E1 334.793} C_DIS
LIN {X -0.098,Y -617.083,Z 1064.656,A 0.000,B 0.000,C 90.000,E1 334.024} C_DIS
LIN {X -0.158,Y -618.504,Z 1064.650,A 0.000,B 0.000,C 90.000,E1 332.999} C_DIS
LIN {X -0.202,Y -619.782,Z 1064.644,A 0.000,B 0.000,C 90.000,E1 331.975} C_DIS
LIN {X 0.054,Y -621.096,Z 1064.637,A 0.000,B 0.000,C 90.000,E1 330.667} C_DIS
LIN {X -0.202,Y -621.844,Z 1064.631,A 0.000,B 0.000,C 90.000,E1 329.665} C_DIS
LIN {X 0.087,Y -622.303,Z 1064.626,A 0.000,B 0.000,C 90.000,E1 328.614} C_DIS
LIN {X 0.176,Y -622.640,Z 1064.620,A 0.000,B 0.000,C 90.000,E1 327.582} C_DIS
LIN {X -0.066,Y -622.594,Z 1064.614,A 0.000,B 0.000,C 90.000,E1 326.580} C_DIS
LIN {X -0.157,Y -622.196,Z 1064.607,A 0.000,B 0.000,C 90.000,E1 325.308} C_DIS
LIN {X -0.069,Y -621.777,Z 1064.602,A 0.000,B 0.000,C 90.000,E1 324.276} C_DIS
LIN {X 0.310,Y -620.750,Z 1064.590,A 0.000,B 0.000,C 90.000,E1 322.190} C_DIS
LIN {X 0.009,Y -619.786,Z 1064.577,A 0.000,B 0.000,C 90.000,E1 319.908} C_DIS
LIN {X 0.323,Y -619.518,Z 1064.572,A 0.000,B 0.000,C 90.000,E1 318.852} C_DIS
LIN {X 0.171,Y -619.138,Z 1064.566,A 0.000,B 0.000,C 90.000,E1 317.838} C_DIS
LIN {X -0.145,Y -618.341,Z 1064.554,A 0.000,B 0.000,C 90.000,E1 315.810} C_DIS
LIN {X -0.192,Y -617.677,Z 1064.546,A 0.000,B 0.000,C 90.000,E1 314.271} C_DIS
LIN {X 0.369,Y -617.477,Z 1064.543,A 0.000,B 0.000,C 90.000,E1 313.704} C_DIS
LIN {X 0.054,Y -617.352,Z 1064.540,A 0.000,B 0.000,C 90.000,E1 313.218} C_DIS
LIN {X 0.167,Y -616.760,Z 1064.533,A 0.000,B 0.000,C 90.000,E1 311.919} C_DIS
LIN {X -0.159,Y -616.478,Z 1064.530,A 0.000,B 0.000,C 90.000,E1 311.434} C_DIS
LIN {X -0.025,Y -616.078,Z 1064.527,A 0.000,B 0.000,C 90.000,E1 310.906} C_DIS
LIN {X 0.273,Y -616.060,Z 1064.526,A 0.000,B 0.000,C 90.000,E1 310.620} C_DIS
LIN {X 0.105,Y -615.792,Z 1064.524,A 0.000,B 0.000,C 90.000,E1 310.378} C_DIS
LIN {X -0.161,Y -615.731,Z 1064.522,A 0.000,B 0.000,C 90.000,E1 309.886} C_DIS
LIN {X -0.046,Y -614.700,Z 1064.510,A 0.000,B 0.000,C 90.000,E1 307.810} C_DIS
LIN {X -0.194,Y -614.394,Z 1064.504,A 0.000,B 0.000,C 90.000,E1 306.790} C_DIS
LIN {X 0.083,Y -613.967,Z 1064.497,A 0.000,B 0.000,C 90.000,E1 305.471} C_DIS
LIN {X 0.175,Y -613.931,Z 1064.494,A 0.000,B 0.000,C 90.000,E1 304.945} C_DIS
LIN {X -0.142,Y -613.509,Z 1064.490,A 0.000,B 0.000,C 90.000,E1 304.199} C_DIS
LIN {X 0.125,Y -613.574,Z 1064.483,A 0.000,B 0.000,C 90.000,E1 302.880} C_DIS
LIN {X -0.024,Y -613.128,Z 1064.473,A 0.000,B 0.000,C 90.000,E1 301.082} C_DIS
LIN {X -0.141,Y -612.561,Z 1064.464,A 0.000,B 0.000,C 90.000,E1 299.539} C_DIS
LIN {X -0.013,Y -611.789,Z 1064.457,A 0.000,B 0.000,C 90.000,E1 298.231} C_DIS
LIN {X 0.093,Y -610.231,Z 1064.450,A 0.000,B 0.000,C 90.000,E1 296.924} C_DIS
LIN {X -0.070,Y -608.394,Z 1064.444,A 0.000,B 0.000,C 90.000,E1 295.899} C_DIS
LIN {X 0.082,Y -606.539,Z 1064.440,A 0.000,B 0.000,C 90.000,E1 295.103} C_DIS
LIN {X -0.017,Y -604.995,Z 1064.437,A 0.000,B 0.000,C 90.000,E1 294.591} C_DIS
LIN {X -0.130,Y -603.122,Z 1064.434,A 0.000,B 0.000,C 90.000,E1 294.079} C_DIS
LIN {X -0.191,Y -602.065,Z 1064.432,A 0.000,B 0.000,C 90.000,E1 293.823} C_DIS
LIN {X 0.221,Y -599.244,Z 1064.429,A 0.000,B 0.000,C 90.000,E1 293.259} C_DIS
LIN {X -0.133,Y -596.798,Z 1064.427,A 0.000,B 0.000,C 90.000,E1 292.898} C_DIS
LIN {X -0.263,Y -593.753,Z 1064.425,A 0.000,B 0.000,C 90.000,E1 292.514} C_DIS
LIN {X -0.026,Y -588.681,Z 1064.422,A 0.000,B 0.000,C 90.000,E1 291.972} C_DIS
LIN {X -0.054,Y -583.479,Z 1064.419,A 0.000,B 0.000,C 90.000,E1 291.461} C_DIS
LIN {X -0.292,Y -574.428,Z 1064.414,A 0.000,B 0.000,C 90.000,E1 290.610} C_DIS
LIN {X -0.173,Y -571.205,Z 1064.413,A 0.000,B 0.000,C 90.000,E1 290.355} C_DIS
LIN {X -0.239,Y -569.461,Z 1064.412,A 0.000,B 0.000,C 90.000,E1 290.248} C_DIS
LIN {X 0.022,Y -567.569,Z 1064.412,A 0.000,B 0.000,C 90.000,E1 290.120} C_DIS
LIN {X 0.120,Y -562.140,Z 1064.411,A 0.000,B 0.000,C 90.000,E1 289.885} C_DIS
LIN {X 0.002,Y -561.508,Z 1064.411,A 0.000,B 0.000,C 90.000,E1 289.885} C_DIS
LIN {X -0.027,Y -546.042,Z 1064.411,A 0.000,B 0.000,C 90.000,E1 289.885} C_DIS
LIN {X 0.206,Y -545.900,Z 1064.410,A 0.000,B 0.000,C 90.000,E1 289.812} C_DIS
LIN {X 0.096,Y -545.753,Z 1064.410,A 0.000,B 0.000,C 90.000,E1 289.704} C_DIS
LIN {X 0.196,Y -544.800,Z 1064.407,A 0.000,B 0.000,C 90.000,E1 289.322} C_DIS
LIN {X 0.283,Y -544.693,Z 1064.406,A 0.000,B 0.000,C 90.000,E1 288.960} C_DIS
LIN {X -0.166,Y -544.395,Z 1064.404,A 0.000,B 0.000,C 90.000,E1 288.725} C_DIS
LIN {X 0.174,Y -544.214,Z 1064.396,A 0.000,B 0.000,C 90.000,E1 287.275} C_DIS
LIN {X -0.176,Y -544.040,Z 1064.388,A 0.000,B 0.000,C 90.000,E1 285.898} C_DIS
LIN {X -0.151,Y -543.675,Z 1064.380,A 0.000,B 0.000,C 90.000,E1 284.481} C_DIS
LIN {X -0.211,Y -543.329,Z 1064.374,A 0.000,B 0.000,C 90.000,E1 283.355} C_DIS
LIN {X 0.128,Y -542.754,Z 1064.368,A 0.000,B 0.000,C 90.000,E1 282.187} C_DIS
LIN {X 0.016,Y -541.944,Z 1064.360,A 0.000,B 0.000,C 90.000,E1 280.782} C_DIS
LIN {X -0.132,Y -541.003,Z 1064.350,A 0.000,B 0.000,C 90.000,E1 279.095} C_DIS
LIN {X 0.155,Y -540.217,Z 1064.343,A 0.000,B 0.000,C 90.000,E1 277.644} C_DIS
LIN {X -0.122,Y -539.030,Z 1064.332,A 0.000,B 0.000,C 90.000,E1 275.682} C_DIS
LIN {X 0.045,Y -538.051,Z 1064.322,A 0.000,B 0.000,C 90.000,E1 273.955} C_DIS
LIN {X 0.104,Y -537.480,Z 1064.316,A 0.000,B 0.000,C 90.000,E1 272.808} C_DIS
LIN {X 0.167,Y -536.534,Z 1064.306,A 0.000,B 0.000,C 90.000,E1 271.088} C_DIS
LIN {X 0.201,Y -535.553,Z 1064.297,A 0.000,B 0.000,C 90.000,E1 269.370} C_DIS
LIN {X 0.225,Y -534.489,Z 1064.287,A 0.000,B 0.000,C 90.000,E1 267.650} C_DIS
LIN {X 0.228,Y -533.624,Z 1064.279,A 0.000,B 0.000,C 90.000,E1 266.216} C_DIS
LIN {X 0.279,Y -532.438,Z 1064.270,A 0.000,B 0.000,C 90.000,E1 264.489} C_DIS
LIN {X -0.227,Y -531.481,Z 1064.263,A 0.000,B 0.000,C 90.000,E1 263.394} C_DIS
LIN {X -0.224,Y -530.320,Z 1064.257,A 0.000,B 0.000,C 90.000,E1 262.243} C_DIS
LIN {X -0.138,Y -527.834,Z 1064.244,A 0.000,B 0.000,C 90.000,E1 259.926} C_DIS
LIN {X -0.011,Y -526.258,Z 1064.236,A 0.000,B 0.000,C 90.000,E1 258.465} C_DIS
LIN {X 0.205,Y -524.761,Z 1064.228,A 0.000,B 0.000,C 90.000,E1 256.992} C_DIS
LIN {X -0.110,Y -523.247,Z 1064.220,A 0.000,B 0.000,C 90.000,E1 255.574} C_DIS
LIN {X 0.182,Y -521.094,Z 1064.208,A 0.000,B 0.000,C 90.000,E1 253.504} C_DIS
LIN {X 0.087,Y -519.600,Z 1064.200,A 0.000,B 0.000,C 90.000,E1 252.054} C_DIS
LIN {X -0.065,Y -517.623,Z 1064.191,A 0.000,B 0.000,C 90.000,E1 250.315} C_DIS
LIN {X -0.055,Y -515.878,Z 1064.182,A 0.000,B 0.000,C 90.000,E1 248.847} C_DIS
LIN {X -0.142,Y -514.690,Z 1064.178,A 0.000,B 0.000,C 90.000,E1 247.975} C_DIS
LIN {X 0.126,Y -512.225,Z 1064.168,A 0.000,B 0.000,C 90.000,E1 246.177} C_DIS
LIN {X -0.031,Y -509.987,Z 1064.160,A 0.000,B 0.000,C 90.000,E1 244.717} C_DIS
LIN {X -0.225,Y -507.599,Z 1064.151,A 0.000,B 0.000,C 90.000,E1 243.256} C_DIS
LIN {X -0.184,Y -506.169,Z 1064.146,A 0.000,B 0.000,C 90.000,E1 242.359} C_DIS
LIN {X 0.079,Y -503.141,Z 1064.136,A 0.000,B 0.000,C 90.000,E1 240.539} C_DIS
LIN {X 0.080,Y -499.860,Z 1064.126,A 0.000,B 0.000,C 90.000,E1 238.742} C_DIS
LIN {X -0.012,Y -497.085,Z 1064.118,A 0.000,B 0.000,C 90.000,E1 237.248} C_DIS
LIN {X 0.263,Y -494.795,Z 1064.111,A 0.000,B 0.000,C 90.000,E1 236.008} C_DIS
LIN {X -0.053,Y -491.865,Z 1064.103,A 0.000,B 0.000,C 90.000,E1 234.529} C_DIS
LIN {X 0.131,Y -489.247,Z 1064.096,A 0.000,B 0.000,C 90.000,E1 233.290} C_DIS
LIN {X -0.223,Y -483.687,Z 1064.083,A 0.000,B 0.000,C 90.000,E1 230.884} C_DIS
LIN {X -0.043,Y -479.566,Z 1064.072,A 0.000,B 0.000,C 90.000,E1 229.013} C_DIS
LIN {X 0.001,Y -475.709,Z 1064.062,A 0.000,B 0.000,C 90.000,E1 227.148} C_DIS
LIN {X 0.044,Y -471.468,Z 1064.050,A 0.000,B 0.000,C 90.000,E1 224.960} C_DIS
LIN {X 0.142,Y -468.495,Z 1064.041,A 0.000,B 0.000,C 90.000,E1 223.380} C_DIS
LIN {X 0.116,Y -466.110,Z 1064.034,A 0.000,B 0.000,C 90.000,E1 222.123} C_DIS
LIN {X -0.106,Y -462.198,Z 1064.024,A 0.000,B 0.000,C 90.000,E1 220.253} C_DIS
LIN {X -0.149,Y -458.972,Z 1064.015,A 0.000,B 0.000,C 90.000,E1 218.669} C_DIS
LIN {X -0.093,Y -455.150,Z 1064.004,A 0.000,B 0.000,C 90.000,E1 216.744} C_DIS
LIN {X 0.160,Y -451.775,Z 1063.995,A 0.000,B 0.000,C 90.000,E1 215.105} C_DIS
LIN {X 0.081,Y -448.361,Z 1063.986,A 0.000,B 0.000,C 90.000,E1 213.499} C_DIS
LIN {X 0.129,Y -444.472,Z 1063.975,A 0.000,B 0.000,C 90.000,E1 211.544} C_DIS
LIN {X 0.033,Y -441.224,Z 1063.966,A 0.000,B 0.000,C 90.000,E1 209.922} C_DIS
LIN {X 0.119,Y -435.278,Z 1063.950,A 0.000,B 0.000,C 90.000,E1 206.950} C_DIS
LIN {X 0.006,Y -431.468,Z 1063.939,A 0.000,B 0.000,C 90.000,E1 204.975} C_DIS
LIN {X -0.069,Y -424.677,Z 1063.917,A 0.000,B 0.000,C 90.000,E1 200.972} C_DIS
LIN {X 0.098,Y -423.255,Z 1063.911,A 0.000,B 0.000,C 90.000,E1 199.939} C_DIS
LIN {X 0.211,Y -421.673,Z 1063.901,A 0.000,B 0.000,C 90.000,E1 198.236} C_DIS
LIN {X -0.189,Y -421.113,Z 1063.896,A 0.000,B 0.000,C 90.000,E1 197.275} C_DIS
LIN {X 0.038,Y -421.180,Z 1063.892,A 0.000,B 0.000,C 90.000,E1 196.567} C_DIS
LIN {X 0.040,Y -421.991,Z 1063.886,A 0.000,B 0.000,C 90.000,E1 195.552} C_DIS
LIN {X -0.128,Y -422.900,Z 1063.883,A 0.000,B 0.000,C 90.000,E1 194.898} C_DIS
LIN {X 0.119,Y -424.419,Z 1063.879,A 0.000,B 0.000,C 90.000,E1 194.189} C_DIS
LIN {X -0.034,Y -426.441,Z 1063.875,A 0.000,B 0.000,C 90.000,E1 193.536} C_DIS
LIN {X -0.078,Y -429.756,Z 1063.871,A 0.000,B 0.000,C 90.000,E1 192.703} C_DIS
LIN {X -0.068,Y -435.560,Z 1063.864,A 0.000,B 0.000,C 90.000,E1 191.535} C_DIS
LIN {X -0.086,Y -445.922,Z 1063.854,A 0.000,B 0.000,C 90.000,E1 189.726} C_DIS
LIN {X 0.125,Y -457.960,Z 1063.843,A 0.000,B 0.000,C 90.000,E1 187.757} C_DIS
LIN {X 0.202,Y -466.854,Z 1063.835,A 0.000,B 0.000,C 90.000,E1 186.315} C_DIS
LIN {X -0.134,Y -471.676,Z 1063.831,A 0.000,B 0.000,C 90.000,E1 185.568} C_DIS
LIN {X 0.215,Y -477.223,Z 1063.826,A 0.000,B 0.000,C 90.000,E1 184.588} C_DIS
LIN {X 0.071,Y -485.257,Z 1063.818,A 0.000,B 0.000,C 90.000,E1 183.212} C_DIS
LIN {X -0.239,Y -494.042,Z 1063.809,A 0.000,B 0.000,C 90.000,E1 181.718} C_DIS
LIN {X -0.115,Y -501.608,Z 1063.802,A 0.000,B 0.000,C 90.000,E1 180.344} C_DIS
LIN {X 0.044,Y -506.623,Z 1063.797,A 0.000,B 0.000,C 90.000,E1 179.427} C_DIS
LIN {X 0.108,Y -514.725,Z 1063.789,A 0.000,B 0.000,C 90.000,E1 177.936} C_DIS
LIN {X 0.122,Y -520.227,Z 1063.783,A 0.000,B 0.000,C 90.000,E1 176.906} C_DIS
LIN {X -0.058,Y -528.091,Z 1063.775,A 0.000,B 0.000,C 90.000,E1 175.469} C_DIS
LIN {X 0.179,Y -535.064,Z 1063.768,A 0.000,B 0.000,C 90.000,E1 174.147} C_DIS
LIN {X -0.139,Y -544.234,Z 1063.758,A 0.000,B 0.000,C 90.000,E1 172.470} C_DIS
LIN {X 0.173,Y -551.602,Z 1063.750,A 0.000,B 0.000,C 90.000,E1 171.027} C_DIS
LIN {X 0.152,Y -558.846,Z 1063.743,A 0.000,B 0.000,C 90.000,E1 169.634} C_DIS
LIN {X 0.199,Y -564.508,Z 1063.736,A 0.000,B 0.000,C 90.000,E1 168.522} C_DIS
LIN {X -0.164,Y -571.919,Z 1063.728,A 0.000,B 0.000,C 90.000,E1 167.048} C_DIS
LIN {X 0.071,Y -577.034,Z 1063.722,A 0.000,B 0.000,C 90.000,E1 165.936} C_DIS
LIN {X 0.179,Y -583.119,Z 1063.714,A 0.000,B 0.000,C 90.000,E1 164.574} C_DIS
LIN {X 0.139,Y -587.804,Z 1063.708,A 0.000,B 0.000,C 90.000,E1 163.504} C_DIS
LIN {X -0.092,Y -591.118,Z 1063.704,A 0.000,B 0.000,C 90.000,E1 162.725} C_DIS
LIN {X 0.150,Y -595.302,Z 1063.698,A 0.000,B 0.000,C 90.000,E1 161.638} C_DIS
LIN {X -0.008,Y -598.259,Z 1063.694,A 0.000,B 0.000,C 90.000,E1 160.859} C_DIS
LIN {X -0.236,Y -602.045,Z 1063.688,A 0.000,B 0.000,C 90.000,E1 159.826} C_DIS
LIN {X -0.202,Y -605.595,Z 1063.682,A 0.000,B 0.000,C 90.000,E1 158.773} C_DIS
LIN {X 0.168,Y -609.723,Z 1063.675,A 0.000,B 0.000,C 90.000,E1 157.433} C_DIS
LIN {X -0.291,Y -613.585,Z 1063.668,A 0.000,B 0.000,C 90.000,E1 156.177} C_DIS
LIN {X 0.155,Y -616.509,Z 1063.662,A 0.000,B 0.000,C 90.000,E1 155.101} C_DIS
LIN {X 0.091,Y -619.223,Z 1063.656,A 0.000,B 0.000,C 90.000,E1 154.076} C_DIS
LIN {X 0.066,Y -622.521,Z 1063.649,A 0.000,B 0.000,C 90.000,E1 152.794} C_DIS
LIN {X 0.076,Y -624.450,Z 1063.645,A 0.000,B 0.000,C 90.000,E1 152.025} C_DIS
LIN {X -0.104,Y -628.115,Z 1063.636,A 0.000,B 0.000,C 90.000,E1 150.511} C_DIS
LIN {X 0.307,Y -631.041,Z 1063.629,A 0.000,B 0.000,C 90.000,E1 149.203} C_DIS
LIN {X -0.325,Y -633.879,Z 1063.622,A 0.000,B 0.000,C 90.000,E1 147.995} C_DIS
LIN {X -0.041,Y -636.604,Z 1063.615,A 0.000,B 0.000,C 90.000,E1 146.707} C_DIS
LIN {X 0.146,Y -639.775,Z 1063.607,A 0.000,B 0.000,C 90.000,E1 145.182} C_DIS
LIN {X -0.128,Y -642.912,Z 1063.598,A 0.000,B 0.000,C 90.000,E1 143.703} C_DIS
LIN {X -0.045,Y -646.567,Z 1063.589,A 0.000,B 0.000,C 90.000,E1 141.949} C_DIS
LIN {X 0.130,Y -650.129,Z 1063.579,A 0.000,B 0.000,C 90.000,E1 140.194} C_DIS
LIN {X -0.078,Y -653.282,Z 1063.571,A 0.000,B 0.000,C 90.000,E1 138.728} C_DIS
LIN {X 0.144,Y -656.488,Z 1063.563,A 0.000,B 0.000,C 90.000,E1 137.229} C_DIS
LIN {X -0.086,Y -661.574,Z 1063.550,A 0.000,B 0.000,C 90.000,E1 135.040} C_DIS
LIN {X -0.163,Y -667.262,Z 1063.538,A 0.000,B 0.000,C 90.000,E1 132.852} C_DIS
LIN {X 0.342,Y -670.505,Z 1063.531,A 0.000,B 0.000,C 90.000,E1 131.595} C_DIS
LIN {X 0.039,Y -674.964,Z 1063.522,A 0.000,B 0.000,C 90.000,E1 129.930} C_DIS
LIN {X -0.216,Y -678.056,Z 1063.515,A 0.000,B 0.000,C 90.000,E1 128.749} C_DIS
LIN {X -0.259,Y -682.422,Z 1063.506,A 0.000,B 0.000,C 90.000,E1 127.076} C_DIS
LIN {X 0.313,Y -686.067,Z 1063.498,A 0.000,B 0.000,C 90.000,E1 125.598} C_DIS
LIN {X -0.218,Y -688.390,Z 1063.493,A 0.000,B 0.000,C 90.000,E1 124.692} C_DIS
LIN {X -0.128,Y -691.318,Z 1063.486,A 0.000,B 0.000,C 90.000,E1 123.499} C_DIS
LIN {X -0.146,Y -694.712,Z 1063.478,A 0.000,B 0.000,C 90.000,E1 122.084} C_DIS
LIN {X -0.095,Y -697.908,Z 1063.470,A 0.000,B 0.000,C 90.000,E1 120.669} C_DIS
LIN {X 0.078,Y -699.379,Z 1063.466,A 0.000,B 0.000,C 90.000,E1 119.951} C_DIS
LIN {X -0.342,Y -700.536,Z 1063.463,A 0.000,B 0.000,C 90.000,E1 119.283} C_DIS
LIN {X -0.413,Y -701.152,Z 1063.460,A 0.000,B 0.000,C 90.000,E1 118.821} C_DIS
LIN {X 0.180,Y -703.364,Z 1063.447,A 0.000,B 0.000,C 90.000,E1 116.437} C_DIS
LIN {X -0.255,Y -704.244,Z 1063.442,A 0.000,B 0.000,C 90.000,E1 115.540} C_DIS
LIN {X -0.036,Y -704.659,Z 1063.438,A 0.000,B 0.000,C 90.000,E1 114.823} C_DIS
LIN {X -0.044,Y -704.688,Z 1063.437,A 0.000,B 0.000,C 90.000,E1 114.591} C_DIS
LIN {X -0.115,Y -704.367,Z 1063.434,A 0.000,B 0.000,C 90.000,E1 114.131} C_DIS
LIN {X -0.117,Y -703.893,Z 1063.433,A 0.000,B 0.000,C 90.000,E1 113.898} C_DIS
LIN {X -0.198,Y -702.509,Z 1063.430,A 0.000,B 0.000,C 90.000,E1 113.439} C_DIS
LIN {X -0.339,Y -701.944,Z 1063.430,A 0.000,B 0.000,C 90.000,E1 113.334} C_DIS
LIN {X 0.204,Y -698.598,Z 1063.427,A 0.000,B 0.000,C 90.000,E1 112.823} C_DIS
LIN {X 0.066,Y -697.621,Z 1063.426,A 0.000,B 0.000,C 90.000,E1 112.717} C_DIS
LIN {X 0.196,Y -696.170,Z 1063.426,A 0.000,B 0.000,C 90.000,E1 112.589} C_DIS
LIN {X 0.000,Y -692.108,Z 1063.425,A 0.000,B 0.000,C 90.000,E1 112.408} C_DIS
LIN {X -0.294,Y -687.044,Z 1063.423,A 0.000,B 0.000,C 90.000,E1 112.206} C_DIS
LIN {X 0.137,Y -684.753,Z 1063.423,A 0.000,B 0.000,C 90.000,E1 112.099} C_DIS
LIN {X -0.334,Y -675.906,Z 1063.422,A 0.000,B 0.000,C 90.000,E1 112.025} C_DIS
LIN {X -0.366,Y -670.073,Z 1063.422,A 0.000,B 0.000,C 90.000,E1 112.025} C_DIS
LIN {X 0.190,Y -608.523,Z 1063.422,A 0.000,B 0.000,C 90.000,E1 111.972} C_DIS
LIN {X 0.221,Y -605.057,Z 1063.422,A 0.000,B 0.000,C 90.000,E1 111.844} C_DIS
LIN {X -0.014,Y -602.741,Z 1063.421,A 0.000,B 0.000,C 90.000,E1 111.770} C_DIS
LIN {X -0.118,Y -597.041,Z 1063.419,A 0.000,B 0.000,C 90.000,E1 111.461} C_DIS
LIN {X 0.129,Y -591.609,Z 1063.417,A 0.000,B 0.000,C 90.000,E1 111.046} C_DIS
LIN {X 0.083,Y -579.703,Z 1063.412,A 0.000,B 0.000,C 90.000,E1 110.066} C_DIS
LIN {X -0.332,Y -575.434,Z 1063.410,A 0.000,B 0.000,C 90.000,E1 109.758} C_DIS
LIN {X 0.036,Y -569.384,Z 1063.407,A 0.000,B 0.000,C 90.000,E1 109.268} C_DIS
LIN {X -0.161,Y -561.031,Z 1063.404,A 0.000,B 0.000,C 90.000,E1 108.779} C_DIS
LIN {X -0.174,Y -554.481,Z 1063.402,A 0.000,B 0.000,C 90.000,E1 108.417} C_DIS
LIN {X 0.023,Y -549.360,Z 1063.400,A 0.000,B 0.000,C 90.000,E1 108.055} C_DIS
LIN {X -0.155,Y -547.696,Z 1063.399,A 0.000,B 0.000,C 90.000,E1 107.873} C_DIS
LIN {X -0.196,Y -547.671,Z 1063.399,A 0.000,B 0.000,C 90.000,E1 107.873} C_DIS
LIN {X 0.200,Y -547.310,Z 1063.397,A 0.000,B 0.000,C 90.000,E1 107.511} C_DIS
LIN {X 0.048,Y -548.652,Z 1063.384,A 0.000,B 0.000,C 90.000,E1 105.134} C_DIS
LIN {X 0.194,Y -550.486,Z 1063.370,A 0.000,B 0.000,C 90.000,E1 102.591} C_DIS
LIN {X 0.029,Y -552.554,Z 1063.358,A 0.000,B 0.000,C 90.000,E1 100.366} C_DIS
LIN {X 0.110,Y -554.375,Z 1063.348,A 0.000,B 0.000,C 90.000,E1 98.681} C_DIS
LIN {X 0.203,Y -556.640,Z 1063.338,A 0.000,B 0.000,C 90.000,E1 96.720} C_DIS
LIN {X 0.031,Y -557.837,Z 1063.331,A 0.000,B 0.000,C 90.000,E1 95.625} C_DIS
LIN {X -0.127,Y -558.890,Z 1063.325,A 0.000,B 0.000,C 90.000,E1 94.531} C_DIS
LIN {X 0.158,Y -559.414,Z 1063.321,A 0.000,B 0.000,C 90.000,E1 93.669} C_DIS
LIN {X -0.199,Y -559.819,Z 1063.318,A 0.000,B 0.000,C 90.000,E1 93.151} C_DIS
LIN {X -0.197,Y -560.634,Z 1063.308,A 0.000,B 0.000,C 90.000,E1 91.489} C_DIS
LIN {X 0.280,Y -561.216,Z 1063.301,A 0.000,B 0.000,C 90.000,E1 90.057} C_DIS
LIN {X -0.144,Y -561.892,Z 1063.290,A 0.000,B 0.000,C 90.000,E1 88.165} C_DIS
LIN {X 0.008,Y -562.615,Z 1063.279,A 0.000,B 0.000,C 90.000,E1 86.216} C_DIS
LIN {X 0.151,Y -563.233,Z 1063.270,A 0.000,B 0.000,C 90.000,E1 84.546} C_DIS
LIN {X -0.244,Y -563.630,Z 1063.261,A 0.000,B 0.000,C 90.000,E1 82.932} C_DIS
LIN {X 0.070,Y -564.222,Z 1063.250,A 0.000,B 0.000,C 90.000,E1 80.971} C_DIS
LIN {X 0.173,Y -565.053,Z 1063.238,A 0.000,B 0.000,C 90.000,E1 78.757} C_DIS
LIN {X 0.076,Y -565.890,Z 1063.229,A 0.000,B 0.000,C 90.000,E1 77.117} C_DIS
LIN {X -0.086,Y -567.166,Z 1063.216,A 0.000,B 0.000,C 90.000,E1 74.936} C_DIS
LIN {X -0.078,Y -568.610,Z 1063.206,A 0.000,B 0.000,C 90.000,E1 73.015} C_DIS
LIN {X 0.321,Y -570.368,Z 1063.193,A 0.000,B 0.000,C 90.000,E1 70.786} C_DIS
LIN {X 0.082,Y -571.536,Z 1063.186,A 0.000,B 0.000,C 90.000,E1 69.444} C_DIS
LIN {X 0.045,Y -573.084,Z 1063.175,A 0.000,B 0.000,C 90.000,E1 67.539} C_DIS
LIN {X 0.052,Y -574.037,Z 1063.168,A 0.000,B 0.000,C 90.000,E1 66.177} C_DIS
LIN {X 0.096,Y -574.572,Z 1063.163,A 0.000,B 0.000,C 90.000,E1 65.357} C_DIS
LIN {X 0.198,Y -575.600,Z 1063.154,A 0.000,B 0.000,C 90.000,E1 63.717} C_DIS
LIN {X 0.056,Y -576.447,Z 1063.145,A 0.000,B 0.000,C 90.000,E1 62.103} C_DIS
LIN {X 0.078,Y -577.181,Z 1063.138,A 0.000,B 0.000,C 90.000,E1 60.745} C_DIS
LIN {X -0.107,Y -577.805,Z 1063.130,A 0.000,B 0.000,C 90.000,E1 59.410} C_DIS
LIN {X -0.128,Y -578.453,Z 1063.121,A 0.000,B 0.000,C 90.000,E1 57.788} C_DIS
LIN {X -0.139,Y -579.171,Z 1063.112,A 0.000,B 0.000,C 90.000,E1 56.167} C_DIS
LIN {X -0.136,Y -579.736,Z 1063.102,A 0.000,B 0.000,C 90.000,E1 54.276} C_DIS
LIN {X -0.281,Y -579.927,Z 1063.095,A 0.000,B 0.000,C 90.000,E1 53.210} C_DIS
LIN {X 0.097,Y -579.960,Z 1063.088,A 0.000,B 0.000,C 90.000,E1 51.823} C_DIS
LIN {X 0.311,Y -579.762,Z 1063.082,A 0.000,B 0.000,C 90.000,E1 50.723} C_DIS
LIN {X 0.114,Y -578.969,Z 1063.072,A 0.000,B 0.000,C 90.000,E1 48.852} C_DIS
LIN {X -0.138,Y -578.443,Z 1063.066,A 0.000,B 0.000,C 90.000,E1 47.796} C_DIS
LIN {X -0.012,Y -577.751,Z 1063.059,A 0.000,B 0.000,C 90.000,E1 46.701} C_DIS
LIN {X -0.032,Y -577.109,Z 1063.055,A 0.000,B 0.000,C 90.000,E1 45.891} C_DIS
LIN {X 0.226,Y -576.638,Z 1063.052,A 0.000,B 0.000,C 90.000,E1 45.324} C_DIS
LIN {X -0.086,Y -575.384,Z 1063.046,A 0.000,B 0.000,C 90.000,E1 44.271} C_DIS
LIN {X 0.000,Y -573.893,Z 1063.040,A 0.000,B 0.000,C 90.000,E1 43.176} C_DIS
LIN {X 0.067,Y -572.241,Z 1063.034,A 0.000,B 0.000,C 90.000,E1 42.081} C_DIS
LIN {X 0.104,Y -570.408,Z 1063.028,A 0.000,B 0.000,C 90.000,E1 40.987} C_DIS
LIN {X 0.048,Y -568.653,Z 1063.023,A 0.000,B 0.000,C 90.000,E1 40.172} C_DIS
LIN {X -0.022,Y -566.743,Z 1063.019,A 0.000,B 0.000,C 90.000,E1 39.358} C_DIS
LIN {X -0.111,Y -564.572,Z 1063.014,A 0.000,B 0.000,C 90.000,E1 38.543} C_DIS
LIN {X -0.226,Y -562.156,Z 1063.010,A 0.000,B 0.000,C 90.000,E1 37.729} C_DIS
LIN {X -0.022,Y -560.407,Z 1063.006,A 0.000,B 0.000,C 90.000,E1 37.156} C_DIS
LIN {X 0.170,Y -558.503,Z 1063.003,A 0.000,B 0.000,C 90.000,E1 36.583} C_DIS
LIN {X 0.347,Y -556.413,Z 1063.000,A 0.000,B 0.000,C 90.000,E1 36.011} C_DIS
LIN {X -0.123,Y -551.748,Z 1062.994,A 0.000,B 0.000,C 90.000,E1 34.945} C_DIS
LIN {X 0.370,Y -547.212,Z 1062.989,A 0.000,B 0.000,C 90.000,E1 33.913} C_DIS
LIN {X 0.047,Y -542.261,Z 1062.983,A 0.000,B 0.000,C 90.000,E1 32.959} C_DIS
LIN {X 0.124,Y -536.909,Z 1062.978,A 0.000,B 0.000,C 90.000,E1 31.957} C_DIS
LIN {X -0.172,Y -531.855,Z 1062.973,A 0.000,B 0.000,C 90.000,E1 31.131} C_DIS
LIN {X 0.114,Y -529.197,Z 1062.970,A 0.000,B 0.000,C 90.000,E1 30.669} C_DIS
LIN {X -0.225,Y -525.356,Z 1062.967,A 0.000,B 0.000,C 90.000,E1 30.129} C_DIS
LIN {X -0.137,Y -521.339,Z 1062.964,A 0.000,B 0.000,C 90.000,E1 29.539} C_DIS
LIN {X -0.077,Y -517.036,Z 1062.961,A 0.000,B 0.000,C 90.000,E1 28.949} C_DIS
LIN {X 0.119,Y -513.631,Z 1062.958,A 0.000,B 0.000,C 90.000,E1 28.487} C_DIS
LIN {X 0.130,Y -508.802,Z 1062.955,A 0.000,B 0.000,C 90.000,E1 27.897} C_DIS
LIN {X -0.048,Y -503.802,Z 1062.952,A 0.000,B 0.000,C 90.000,E1 27.334} C_DIS
LIN {X 0.133,Y -499.784,Z 1062.949,A 0.000,B 0.000,C 90.000,E1 26.873} C_DIS
LIN {X -0.097,Y -490.424,Z 1062.944,A 0.000,B 0.000,C 90.000,E1 25.924} C_DIS
LIN {X -0.108,Y -479.138,Z 1062.938,A 0.000,B 0.000,C 90.000,E1 24.823} C_DIS
LIN {X -0.182,Y -469.132,Z 1062.933,A 0.000,B 0.000,C 90.000,E1 23.898} C_DIS
LIN {X 0.207,Y -458.716,Z 1062.928,A 0.000,B 0.000,C 90.000,E1 22.950} C_DIS
LIN {X -0.101,Y -446.860,Z 1062.922,A 0.000,B 0.000,C 90.000,E1 21.972} C_DIS
LIN {X -0.104,Y -429.150,Z 1062.913,A 0.000,B 0.000,C 90.000,E1 20.355} C_DIS
LIN {X -0.120,Y -416.174,Z 1062.906,A 0.000,B 0.000,C 90.000,E1 19.033} C_DIS
LIN {X 0.174,Y -403.929,Z 1062.898,A 0.000,B 0.000,C 90.000,E1 17.583} C_DIS
LIN {X 0.044,Y -399.956,Z 1062.895,A 0.000,B 0.000,C 90.000,E1 17.094} C_DIS
LIN {X 0.093,Y -395.421,Z 1062.891,A 0.000,B 0.000,C 90.000,E1 16.386} C_DIS
LIN {X 0.061,Y -393.399,Z 1062.889,A 0.000,B 0.000,C 90.000,E1 15.969} C_DIS
LIN {X 0.092,Y -392.760,Z 1062.888,A 0.000,B 0.000,C 90.000,E1 15.788} C_DIS
LIN {X -0.102,Y -391.950,Z 1062.886,A 0.000,B 0.000,C 90.000,E1 15.426} C_DIS
LIN {X 0.005,Y -391.656,Z 1062.883,A 0.000,B 0.000,C 90.000,E1 14.898} C_DIS
LIN {X -0.006,Y -391.924,Z 1062.879,A 0.000,B 0.000,C 90.000,E1 14.189} C_DIS
LIN {X 0.035,Y -392.192,Z 1062.877,A 0.000,B 0.000,C 90.000,E1 13.828} C_DIS
LIN {X -0.194,Y -398.943,Z 1062.851,A 0.000,B 0.000,C 90.000,E1 9.265} C_DIS
LIN {X 0.133,Y -401.503,Z 1062.844,A 0.000,B 0.000,C 90.000,E1 7.814} C_DIS
LIN {X -0.050,Y -409.042,Z 1062.824,A 0.000,B 0.000,C 90.000,E1 4.359} C_DIS
LIN {X -0.063,Y -411.564,Z 1062.819,A 0.000,B 0.000,C 90.000,E1 3.498} C_DIS
LIN {X -0.071,Y -413.702,Z 1062.818,A 0.000,B 0.000,C 90.000,E1 3.154} C_DIS
LIN {X -0.048,Y -415.965,Z 1062.816,A 0.000,B 0.000,C 90.000,E1 2.808} C_DIS
LIN {X -0.046,Y -417.266,Z 1062.815,A 0.000,B 0.000,C 90.000,E1 2.636} C_DIS
LIN {X -0.194,Y -422.846,Z 1062.812,A 0.000,B 0.000,C 90.000,E1 2.178} C_DIS
LIN {X 0.066,Y -434.766,Z 1062.808,A 0.000,B 0.000,C 90.000,E1 1.375} C_DIS
LIN {X -0.010,Y -454.612,Z 1062.801,A 0.000,B 0.000,C 90.000,E1 0.115} C_DIS
LIN {X -0.153,Y -469.717,Z 1062.796,A 0.000,B 0.000,C 90.000,E1 359.198} C_DIS
LIN {X 0.186,Y -485.914,Z 1062.790,A 0.000,B 0.000,C 90.000,E1 358.165} C_DIS
LIN {X 0.019,Y -496.980,Z 1062.786,A 0.000,B 0.000,C 90.000,E1 357.478} C_DIS
LIN {X -0.066,Y -504.740,Z 1062.783,A 0.000,B 0.000,C 90.000,E1 356.963} C_DIS
LIN {X 0.098,Y -510.911,Z 1062.781,A 0.000,B 0.000,C 90.000,E1 356.502} C_DIS
LIN {X 0.067,Y -516.944,Z 1062.778,A 0.000,B 0.000,C 90.000,E1 356.045} C_DIS
LIN {X 0.074,Y -522.619,Z 1062.776,A 0.000,B 0.000,C 90.000,E1 355.584} C_DIS
LIN {X -0.069,Y -529.373,Z 1062.772,A 0.000,B 0.000,C 90.000,E1 355.008} C_DIS
LIN {X -0.219,Y -536.101,Z 1062.769,A 0.000,B 0.000,C 90.000,E1 354.375} C_DIS
LIN {X -0.170,Y -542.458,Z 1062.765,A 0.000,B 0.000,C 90.000,E1 353.685} C_DIS
LIN {X 0.089,Y -547.251,Z 1062.762,A 0.000,B 0.000,C 90.000,E1 353.109} C_DIS
LIN {X 0.130,Y -552.485,Z 1062.758,A 0.000,B 0.000,C 90.000,E1 352.413} C_DIS
LIN {X -0.196,Y -556.373,Z 1062.755,A 0.000,B 0.000,C 90.000,E1 351.894} C_DIS
LIN {X -0.179,Y -560.736,Z 1062.751,A 0.000,B 0.000,C 90.000,E1 351.197} C_DIS
LIN {X 0.030,Y -564.001,Z 1062.748,A 0.000,B 0.000,C 90.000,E1 350.622} C_DIS
LIN {X 0.112,Y -567.652,Z 1062.744,A 0.000,B 0.000,C 90.000,E1 349.926} C_DIS
LIN {X -0.094,Y -570.373,Z 1062.741,A 0.000,B 0.000,C 90.000,E1 349.398} C_DIS
LIN {X 0.119,Y -575.390,Z 1062.735,A 0.000,B 0.000,C 90.000,E1 348.285} C_DIS
LIN {X -0.166,Y -579.971,Z 1062.729,A 0.000,B 0.000,C 90.000,E1 347.229} C_DIS
LIN {X 0.173,Y -584.223,Z 1062.723,A 0.000,B 0.000,C 90.000,E1 346.117} C_DIS
LIN {X -0.177,Y -589.166,Z 1062.716,A 0.000,B 0.000,C 90.000,E1 344.810} C_DIS
LIN {X 0.174,Y -592.099,Z 1062.711,A 0.000,B 0.000,C 90.000,E1 343.976} C_DIS
LIN {X -0.047,Y -596.745,Z 1062.704,A 0.000,B 0.000,C 90.000,E1 342.670} C_DIS
LIN {X 0.170,Y -601.003,Z 1062.696,A 0.000,B 0.000,C 90.000,E1 341.329} C_DIS
LIN {X -0.014,Y -604.021,Z 1062.691,A 0.000,B 0.000,C 90.000,E1 340.296} C_DIS
LIN {X -0.159,Y -606.846,Z 1062.685,A 0.000,B 0.000,C 90.000,E1 339.263} C_DIS
LIN {X 0.235,Y -610.154,Z 1062.677,A 0.000,B 0.000,C 90.000,E1 337.922} C_DIS
LIN {X -0.217,Y -613.058,Z 1062.670,A 0.000,B 0.000,C 90.000,E1 336.666} C_DIS
LIN {X -0.029,Y -615.061,Z 1062.665,A 0.000,B 0.000,C 90.000,E1 335.613} C_DIS
LIN {X -0.120,Y -616.797,Z 1062.659,A 0.000,B 0.000,C 90.000,E1 334.588} C_DIS
LIN {X -0.168,Y -617.887,Z 1062.655,A 0.000,B 0.000,C 90.000,E1 333.819} C_DIS
LIN {X -0.213,Y -619.311,Z 1062.649,A 0.000,B 0.000,C 90.000,E1 332.794} C_DIS
LIN {X -0.243,Y -620.560,Z 1062.643,A 0.000,B 0.000,C 90.000,E1 331.769} C_DIS
LIN {X 0.036,Y -621.656,Z 1062.637,A 0.000,B 0.000,C 90.000,E1 330.717} C_DIS
LIN {X 0.330,Y -622.465,Z 1062.632,A 0.000,B 0.000,C 90.000,E1 329.665} C_DIS
LIN {X 0.089,Y -623.069,Z 1062.625,A 0.000,B 0.000,C 90.000,E1 328.408} C_DIS
LIN {X 0.192,Y -623.415,Z 1062.619,A 0.000,B 0.000,C 90.000,E1 327.375} C_DIS
LIN {X -0.041,Y -623.380,Z 1062.613,A 0.000,B 0.000,C 90.000,E1 326.373} C_DIS
LIN {X 0.062,Y -623.126,Z 1062.608,A 0.000,B 0.000,C 90.000,E1 325.341} C_DIS
LIN {X 0.012,Y -622.821,Z 1062.602,A 0.000,B 0.000,C 90.000,E1 324.322} C_DIS
LIN {X 0.053,Y -621.921,Z 1062.590,A 0.000,B 0.000,C 90.000,E1 322.271} C_DIS
LIN {X -0.202,Y -620.942,Z 1062.573,A 0.000,B 0.000,C 90.000,E1 319.218} C_DIS
LIN {X 0.130,Y -620.679,Z 1062.568,A 0.000,B 0.000,C 90.000,E1 318.162} C_DIS
LIN {X 0.149,Y -620.049,Z 1062.559,A 0.000,B 0.000,C 90.000,E1 316.620} C_DIS
LIN {X -0.003,Y -619.757,Z 1062.553,A 0.000,B 0.000,C 90.000,E1 315.607} C_DIS
LIN {X -0.043,Y -619.091,Z 1062.541,A 0.000,B 0.000,C 90.000,E1 313.299} C_DIS
LIN {X -0.056,Y -618.514,Z 1062.532,A 0.000,B 0.000,C 90.000,E1 311.757} C_DIS
LIN {X -0.341,Y -617.457,Z 1062.521,A 0.000,B 0.000,C 90.000,E1 309.725} C_DIS
LIN {X -0.125,Y -616.413,Z 1062.505,A 0.000,B 0.000,C 90.000,E1 306.870} C_DIS
LIN {X -0.254,Y -615.930,Z 1062.493,A 0.000,B 0.000,C 90.000,E1 304.818} C_DIS
LIN {X 0.016,Y -615.844,Z 1062.485,A 0.000,B 0.000,C 90.000,E1 303.245} C_DIS
LIN {X 0.057,Y -615.710,Z 1062.480,A 0.000,B 0.000,C 90.000,E1 302.467} C_DIS
LIN {X -0.009,Y -615.760,Z 1062.478,A 0.000,B 0.000,C 90.000,E1 301.957} C_DIS
LIN {X -0.039,Y -615.489,Z 1062.470,A 0.000,B 0.000,C 90.000,E1 300.669} C_DIS
LIN {X -0.066,Y -615.361,Z 1062.469,A 0.000,B 0.000,C 90.000,E1 300.413} C_DIS
LIN {X 0.219,Y -615.461,Z 1062.468,A 0.000,B 0.000,C 90.000,E1 300.129} C_DIS
LIN {X -0.116,Y -615.197,Z 1062.462,A 0.000,B 0.000,C 90.000,E1 299.127} C_DIS
LIN {X -0.142,Y -615.304,Z 1062.460,A 0.000,B 0.000,C 90.000,E1 298.871} C_DIS
LIN {X -0.189,Y -615.068,Z 1062.458,A 0.000,B 0.000,C 90.000,E1 298.359} C_DIS
LIN {X 0.002,Y -614.464,Z 1062.452,A 0.000,B 0.000,C 90.000,E1 297.308} C_DIS
LIN {X -0.104,Y -613.329,Z 1062.446,A 0.000,B 0.000,C 90.000,E1 296.283} C_DIS
LIN {X 0.328,Y -611.678,Z 1062.440,A 0.000,B 0.000,C 90.000,E1 295.207} C_DIS
LIN {X -0.035,Y -610.078,Z 1062.436,A 0.000,B 0.000,C 90.000,E1 294.463} C_DIS
LIN {X -0.161,Y -607.768,Z 1062.432,A 0.000,B 0.000,C 90.000,E1 293.695} C_DIS
LIN {X 0.057,Y -605.846,Z 1062.429,A 0.000,B 0.000,C 90.000,E1 293.153} C_DIS
LIN {X -0.057,Y -603.285,Z 1062.426,A 0.000,B 0.000,C 90.000,E1 292.642} C_DIS
LIN {X -0.124,Y -601.690,Z 1062.424,A 0.000,B 0.000,C 90.000,E1 292.386} C_DIS
LIN {X 0.133,Y -599.969,Z 1062.423,A 0.000,B 0.000,C 90.000,E1 292.099} C_DIS
LIN {X 0.013,Y -597.019,Z 1062.421,A 0.000,B 0.000,C 90.000,E1 291.716} C_DIS
LIN {X 0.208,Y -590.694,Z 1062.417,A 0.000,B 0.000,C 90.000,E1 291.046} C_DIS
LIN {X 0.177,Y -587.859,Z 1062.416,A 0.000,B 0.000,C 90.000,E1 290.791} C_DIS
LIN {X 0.256,Y -586.345,Z 1062.415,A 0.000,B 0.000,C 90.000,E1 290.663} C_DIS
LIN {X 0.129,Y -582.388,Z 1062.413,A 0.000,B 0.000,C 90.000,E1 290.301} C_DIS
LIN {X 0.180,Y -580.487,Z 1062.412,A 0.000,B 0.000,C 90.000,E1 290.174} C_DIS
LIN {X -0.023,Y -576.778,Z 1062.411,A 0.000,B 0.000,C 90.000,E1 289.885} C_DIS
LIN {X 0.097,Y -571.818,Z 1062.409,A 0.000,B 0.000,C 90.000,E1 289.631} C_DIS
LIN {X -0.018,Y -569.521,Z 1062.408,A 0.000,B 0.000,C 90.000,E1 289.504} C_DIS
LIN {X 0.111,Y -567.586,Z 1062.408,A 0.000,B 0.000,C 90.000,E1 289.396} C_DIS
LIN {X -0.226,Y -559.516,Z 1062.407,A 0.000,B 0.000,C 90.000,E1 289.214} C_DIS
LIN {X -0.262,Y -546.182,Z 1062.407,A 0.000,B 0.000,C 90.000,E1 289.214} C_DIS
LIN {X -0.020,Y -545.685,Z 1062.406,A 0.000,B 0.000,C 90.000,E1 289.087} C_DIS
LIN {X -0.062,Y -545.661,Z 1062.406,A 0.000,B 0.000,C 90.000,E1 289.087} C_DIS
LIN {X -0.129,Y -545.208,Z 1062.405,A 0.000,B 0.000,C 90.000,E1 288.852} C_DIS
LIN {X -0.054,Y -544.564,Z 1062.395,A 0.000,B 0.000,C 90.000,E1 287.149} C_DIS
LIN {X 0.120,Y -544.318,Z 1062.387,A 0.000,B 0.000,C 90.000,E1 285.717} C_DIS
LIN {X 0.149,Y -543.960,Z 1062.380,A 0.000,B 0.000,C 90.000,E1 284.300} C_DIS
LIN {X 0.088,Y -543.578,Z 1062.373,A 0.000,B 0.000,C 90.000,E1 283.175} C_DIS
LIN {X 0.066,Y -542.670,Z 1062.364,A 0.000,B 0.000,C 90.000,E1 281.478} C_DIS
LIN {X 0.007,Y -541.516,Z 1062.353,A 0.000,B 0.000,C 90.000,E1 279.500} C_DIS
LIN {X -0.231,Y -540.721,Z 1062.345,A 0.000,B 0.000,C 90.000,E1 278.106} C_DIS
LIN {X 0.039,Y -539.686,Z 1062.335,A 0.000,B 0.000,C 90.000,E1 276.372} C_DIS
LIN {X 0.170,Y -538.877,Z 1062.328,A 0.000,B 0.000,C 90.000,E1 274.935} C_DIS
LIN {X -0.201,Y -537.798,Z 1062.317,A 0.000,B 0.000,C 90.000,E1 272.980} C_DIS
LIN {X -0.132,Y -536.850,Z 1062.307,A 0.000,B 0.000,C 90.000,E1 271.260} C_DIS
LIN {X -0.087,Y -535.694,Z 1062.296,A 0.000,B 0.000,C 90.000,E1 269.255} C_DIS
LIN {X -0.061,Y -534.618,Z 1062.286,A 0.000,B 0.000,C 90.000,E1 267.535} C_DIS
LIN {X -0.048,Y -533.935,Z 1062.280,A 0.000,B 0.000,C 90.000,E1 266.388} C_DIS
LIN {X -0.037,Y -532.746,Z 1062.270,A 0.000,B 0.000,C 90.000,E1 264.666} C_DIS
LIN {X -0.017,Y -531.811,Z 1062.264,A 0.000,B 0.000,C 90.000,E1 263.514} C_DIS
LIN {X 0.055,Y -530.695,Z 1062.258,A 0.000,B 0.000,C 90.000,E1 262.356} C_DIS
LIN {X 0.185,Y -527.916,Z 1062.243,A 0.000,B 0.000,C 90.000,E1 259.746} C_DIS
LIN {X -0.149,Y -525.736,Z 1062.232,A 0.000,B 0.000,C 90.000,E1 257.757} C_DIS
LIN {X 0.088,Y -523.589,Z 1062.221,A 0.000,B 0.000,C 90.000,E1 255.700} C_DIS
LIN {X -0.118,Y -521.439,Z 1062.209,A 0.000,B 0.000,C 90.000,E1 253.685} C_DIS
LIN {X -0.208,Y -519.952,Z 1062.201,A 0.000,B 0.000,C 90.000,E1 252.236} C_DIS
LIN {X 0.311,Y -518.010,Z 1062.192,A 0.000,B 0.000,C 90.000,E1 250.423} C_DIS
LIN {X -0.198,Y -515.873,Z 1062.182,A 0.000,B 0.000,C 90.000,E1 248.720} C_DIS
LIN {X -0.154,Y -514.242,Z 1062.175,A 0.000,B 0.000,C 90.000,E1 247.539} C_DIS
LIN {X -0.012,Y -512.217,Z 1062.167,A 0.000,B 0.000,C 90.000,E1 246.049} C_DIS
LIN {X -0.167,Y -509.950,Z 1062.159,A 0.000,B 0.000,C 90.000,E1 244.588} C_DIS
LIN {X 0.091,Y -507.560,Z 1062.151,A 0.000,B 0.000,C 90.000,E1 243.076} C_DIS
LIN {X -0.321,Y -506.117,Z 1062.146,A 0.000,B 0.000,C 90.000,E1 242.231} C_DIS
LIN {X -0.060,Y -503.085,Z 1062.136,A 0.000,B 0.000,C 90.000,E1 240.411} C_DIS
LIN {X -0.062,Y -499.754,Z 1062.126,A 0.000,B 0.000,C 90.000,E1 238.614} C_DIS
LIN {X -0.157,Y -496.985,Z 1062.117,A 0.000,B 0.000,C 90.000,E1 237.120} C_DIS
LIN {X 0.114,Y -494.685,Z 1062.111,A 0.000,B 0.000,C 90.000,E1 235.881} C_DIS
LIN {X -0.206,Y -491.742,Z 1062.102,A 0.000,B 0.000,C 90.000,E1 234.402} C_DIS
LIN {X -0.263,Y -489.751,Z 1062.097,A 0.000,B 0.000,C 90.000,E1 233.497} C_DIS
LIN {X 0.087,Y -484.163,Z 1062.083,A 0.000,B 0.000,C 90.000,E1 231.009} C_DIS
LIN {X 0.161,Y -480.685,Z 1062.075,A 0.000,B 0.000,C 90.000,E1 229.461} C_DIS
LIN {X -0.090,Y -476.775,Z 1062.065,A 0.000,B 0.000,C 90.000,E1 227.634} C_DIS
LIN {X -0.261,Y -471.855,Z 1062.051,A 0.000,B 0.000,C 90.000,E1 225.162} C_DIS
LIN {X 0.096,Y -469.468,Z 1062.044,A 0.000,B 0.000,C 90.000,E1 223.866} C_DIS
LIN {X 0.158,Y -466.470,Z 1062.035,A 0.000,B 0.000,C 90.000,E1 222.285} C_DIS
LIN {X -0.055,Y -462.559,Z 1062.025,A 0.000,B 0.000,C 90.000,E1 220.415} C_DIS
LIN {X -0.087,Y -459.310,Z 1062.016,A 0.000,B 0.000,C 90.000,E1 218.830} C_DIS
LIN {X -0.017,Y -454.836,Z 1062.003,A 0.000,B 0.000,C 90.000,E1 216.583} C_DIS
LIN {X -0.035,Y -451.444,Z 1061.994,A 0.000,B 0.000,C 90.000,E1 214.978} C_DIS
LIN {X -0.041,Y -447.337,Z 1061.984,A 0.000,B 0.000,C 90.000,E1 213.038} C_DIS
LIN {X -0.070,Y -444.065,Z 1061.974,A 0.000,B 0.000,C 90.000,E1 211.416} C_DIS
LIN {X -0.171,Y -440.773,Z 1061.965,A 0.000,B 0.000,C 90.000,E1 209.795} C_DIS
LIN {X 0.101,Y -434.794,Z 1061.949,A 0.000,B 0.000,C 90.000,E1 206.796} C_DIS
LIN {X -0.040,Y -430.869,Z 1061.938,A 0.000,B 0.000,C 90.000,E1 204.823} C_DIS
LIN {X 0.089,Y -425.046,Z 1061.919,A 0.000,B 0.000,C 90.000,E1 201.461} C_DIS
LIN {X -0.165,Y -422.608,Z 1061.910,A 0.000,B 0.000,C 90.000,E1 199.812} C_DIS
LIN {X -0.068,Y -421.016,Z 1061.901,A 0.000,B 0.000,C 90.000,E1 198.109} C_DIS
LIN {X -0.077,Y -420.388,Z 1061.895,A 0.000,B 0.000,C 90.000,E1 197.094} C_DIS
LIN {X 0.145,Y -420.364,Z 1061.891,A 0.000,B 0.000,C 90.000,E1 196.386} C_DIS
LIN {X 0.137,Y -420.991,Z 1061.885,A 0.000,B 0.000,C 90.000,E1 195.371} C_DIS
LIN {X -0.040,Y -421.771,Z 1061.882,A 0.000,B 0.000,C 90.000,E1 194.717} C_DIS
LIN {X -0.213,Y -423.205,Z 1061.878,A 0.000,B 0.000,C 90.000,E1 194.064} C_DIS
LIN {X 0.035,Y -425.155,Z 1061.874,A 0.000,B 0.000,C 90.000,E1 193.355} C_DIS
LIN {X -0.117,Y -428.420,Z 1061.870,A 0.000,B 0.000,C 90.000,E1 192.535} C_DIS
LIN {X -0.189,Y -434.043,Z 1061.863,A 0.000,B 0.000,C 90.000,E1 191.422} C_DIS
LIN {X 0.039,Y -442.594,Z 1061.855,A 0.000,B 0.000,C 90.000,E1 189.905} C_DIS
LIN {X 0.182,Y -454.719,Z 1061.844,A 0.000,B 0.000,C 90.000,E1 187.936} C_DIS
LIN {X -0.065,Y -460.811,Z 1061.839,A 0.000,B 0.000,C 90.000,E1 187.004} C_DIS
LIN {X -0.210,Y -467.803,Z 1061.833,A 0.000,B 0.000,C 90.000,E1 185.910} C_DIS
LIN {X -0.072,Y -472.617,Z 1061.828,A 0.000,B 0.000,C 90.000,E1 185.106} C_DIS
LIN {X 0.117,Y -477.268,Z 1061.824,A 0.000,B 0.000,C 90.000,E1 184.302} C_DIS
LIN {X -0.145,Y -484.519,Z 1061.817,A 0.000,B 0.000,C 90.000,E1 183.094} C_DIS
LIN {X -0.172,Y -492.548,Z 1061.809,A 0.000,B 0.000,C 90.000,E1 181.718} C_DIS
LIN {X -0.075,Y -500.292,Z 1061.802,A 0.000,B 0.000,C 90.000,E1 180.344} C_DIS
LIN {X -0.039,Y -506.937,Z 1061.795,A 0.000,B 0.000,C 90.000,E1 179.141} C_DIS
LIN {X -0.188,Y -514.304,Z 1061.788,A 0.000,B 0.000,C 90.000,E1 177.822} C_DIS
LIN {X -0.215,Y -521.451,Z 1061.781,A 0.000,B 0.000,C 90.000,E1 176.502} C_DIS
LIN {X 0.150,Y -527.779,Z 1061.774,A 0.000,B 0.000,C 90.000,E1 175.298} C_DIS
LIN {X 0.124,Y -534.031,Z 1061.768,A 0.000,B 0.000,C 90.000,E1 174.147} C_DIS
LIN {X -0.215,Y -543.213,Z 1061.758,A 0.000,B 0.000,C 90.000,E1 172.470} C_DIS
LIN {X 0.077,Y -550.683,Z 1061.750,A 0.000,B 0.000,C 90.000,E1 171.027} C_DIS
LIN {X -0.253,Y -557.241,Z 1061.743,A 0.000,B 0.000,C 90.000,E1 169.803} C_DIS
LIN {X -0.083,Y -562.267,Z 1061.738,A 0.000,B 0.000,C 90.000,E1 168.814} C_DIS
LIN {X 0.148,Y -567.049,Z 1061.733,A 0.000,B 0.000,C 90.000,E1 167.825} C_DIS
LIN {X -0.118,Y -572.452,Z 1061.726,A 0.000,B 0.000,C 90.000,E1 166.756} C_DIS
LIN {X -0.084,Y -576.316,Z 1061.722,A 0.000,B 0.000,C 90.000,E1 165.936} C_DIS
LIN {X -0.082,Y -583.079,Z 1061.714,A 0.000,B 0.000,C 90.000,E1 164.448} C_DIS
LIN {X -0.120,Y -587.747,Z 1061.708,A 0.000,B 0.000,C 90.000,E1 163.378} C_DIS
LIN {X -0.103,Y -592.138,Z 1061.702,A 0.000,B 0.000,C 90.000,E1 162.308} C_DIS
LIN {X 0.150,Y -596.265,Z 1061.696,A 0.000,B 0.000,C 90.000,E1 161.221} C_DIS
LIN {X -0.196,Y -601.102,Z 1061.688,A 0.000,B 0.000,C 90.000,E1 159.934} C_DIS
LIN {X 0.180,Y -604.714,Z 1061.683,A 0.000,B 0.000,C 90.000,E1 158.847} C_DIS
LIN {X 0.199,Y -608.928,Z 1061.675,A 0.000,B 0.000,C 90.000,E1 157.539} C_DIS
LIN {X -0.225,Y -612.067,Z 1061.670,A 0.000,B 0.000,C 90.000,E1 156.538} C_DIS
LIN {X -0.076,Y -615.772,Z 1061.662,A 0.000,B 0.000,C 90.000,E1 155.229} C_DIS
LIN {X -0.152,Y -618.521,Z 1061.657,A 0.000,B 0.000,C 90.000,E1 154.204} C_DIS
LIN {X -0.182,Y -620.561,Z 1061.652,A 0.000,B 0.000,C 90.000,E1 153.435} C_DIS
LIN {X -0.190,Y -623.182,Z 1061.647,A 0.000,B 0.000,C 90.000,E1 152.410} C_DIS
LIN {X 0.166,Y -627.483,Z 1061.637,A 0.000,B 0.000,C 90.000,E1 150.589} C_DIS
LIN {X 0.041,Y -631.052,Z 1061.628,A 0.000,B 0.000,C 90.000,E1 149.076} C_DIS
LIN {X -0.233,Y -634.399,Z 1061.620,A 0.000,B 0.000,C 90.000,E1 147.582} C_DIS
LIN {X 0.062,Y -637.107,Z 1061.613,A 0.000,B 0.000,C 90.000,E1 146.294} C_DIS
LIN {X 0.259,Y -640.307,Z 1061.604,A 0.000,B 0.000,C 90.000,E1 144.769} C_DIS
LIN {X -0.036,Y -642.919,Z 1061.598,A 0.000,B 0.000,C 90.000,E1 143.543} C_DIS
LIN {X 0.142,Y -646.118,Z 1061.589,A 0.000,B 0.000,C 90.000,E1 142.029} C_DIS
LIN {X 0.305,Y -649.703,Z 1061.579,A 0.000,B 0.000,C 90.000,E1 140.275} C_DIS
LIN {X -0.403,Y -652.888,Z 1061.571,A 0.000,B 0.000,C 90.000,E1 138.852} C_DIS
LIN {X 0.264,Y -656.626,Z 1061.562,A 0.000,B 0.000,C 90.000,E1 137.067} C_DIS
LIN {X 0.060,Y -661.158,Z 1061.551,A 0.000,B 0.000,C 90.000,E1 135.121} C_DIS
LIN {X -0.028,Y -666.890,Z 1061.539,A 0.000,B 0.000,C 90.000,E1 132.933} C_DIS
LIN {X 0.026,Y -670.143,Z 1061.532,A 0.000,B 0.000,C 90.000,E1 131.714} C_DIS
LIN {X 0.165,Y -674.598,Z 1061.522,A 0.000,B 0.000,C 90.000,E1 130.011} C_DIS
LIN {X -0.077,Y -678.361,Z 1061.514,A 0.000,B 0.000,C 90.000,E1 128.588} C_DIS
LIN {X -0.140,Y -682.082,Z 1061.506,A 0.000,B 0.000,C 90.000,E1 127.156} C_DIS
LIN {X -0.127,Y -685.759,Z 1061.498,A 0.000,B 0.000,C 90.000,E1 125.724} C_DIS
LIN {X 0.290,Y -688.092,Z 1061.493,A 0.000,B 0.000,C 90.000,E1 124.739} C_DIS
LIN {X -0.013,Y -691.032,Z 1061.487,A 0.000,B 0.000,C 90.000,E1 123.579} C_DIS
LIN {X 0.339,Y -694.417,Z 1061.479,A 0.000,B 0.000,C 90.000,E1 122.133} C_DIS
LIN {X 0.021,Y -697.646,Z 1061.471,A 0.000,B 0.000,C 90.000,E1 120.747} C_DIS
LIN {X -0.062,Y -699.123,Z 1061.467,A 0.000,B 0.000,C 90.000,E1 120.050} C_DIS
LIN {X 0.119,Y -700.342,Z 1061.463,A 0.000,B 0.000,C 90.000,E1 119.333} C_DIS
LIN {X 0.313,Y -701.195,Z 1061.459,A 0.000,B 0.000,C 90.000,E1 118.615} C_DIS
LIN {X -0.010,Y -703.205,Z 1061.448,A 0.000,B 0.000,C 90.000,E1 116.539} C_DIS
LIN {X 0.178,Y -704.099,Z 1061.442,A 0.000,B 0.000,C 90.000,E1 115.591} C_DIS
LIN {X 0.096,Y -704.557,Z 1061.438,A 0.000,B 0.000,C 90.000,E1 114.899} C_DIS
LIN {X 0.383,Y -704.674,Z 1061.437,A 0.000,B 0.000,C 90.000,E1 114.643} C_DIS
LIN {X 0.020,Y -704.387,Z 1061.435,A 0.000,B 0.000,C 90.000,E1 114.207} C_DIS
LIN {X 0.305,Y -704.115,Z 1061.433,A 0.000,B 0.000,C 90.000,E1 113.951} C_DIS
LIN {X -0.058,Y -702.775,Z 1061.431,A 0.000,B 0.000,C 90.000,E1 113.515} C_DIS
LIN {X 0.219,Y -701.754,Z 1061.429,A 0.000,B 0.000,C 90.000,E1 113.259} C_DIS
LIN {X -0.158,Y -698.414,Z 1061.427,A 0.000,B 0.000,C 90.000,E1 112.823} C_DIS
LIN {X -0.028,Y -697.346,Z 1061.426,A 0.000,B 0.000,C 90.000,E1 112.695} C_DIS
LIN {X -0.166,Y -695.728,Z 1061.425,A 0.000,B 0.000,C 90.000,E1 112.589} C_DIS
LIN {X 0.265,Y -688.250,Z 1061.424,A 0.000,B 0.000,C 90.000,E1 112.206} C_DIS
LIN {X 0.011,Y -686.302,Z 1061.423,A 0.000,B 0.000,C 90.000,E1 112.153} C_DIS
LIN {X 0.017,Y -682.922,Z 1061.423,A 0.000,B 0.000,C 90.000,E1 112.078} C_DIS
LIN {X -0.343,Y -676.272,Z 1061.422,A 0.000,B 0.000,C 90.000,E1 112.025} C_DIS
LIN {X 0.198,Y -608.886,Z 1061.422,A 0.000,B 0.000,C 90.000,E1 111.972} C_DIS
LIN {X -0.114,Y -604.571,Z 1061.421,A 0.000,B 0.000,C 90.000,E1 111.844} C_DIS
LIN {X 0.178,Y -602.281,Z 1061.421,A 0.000,B 0.000,C 90.000,E1 111.716} C_DIS
LIN {X -0.072,Y -597.268,Z 1061.419,A 0.000,B 0.000,C 90.000,E1 111.461} C_DIS
LIN {X 0.196,Y -590.858,Z 1061.417,A 0.000,B 0.000,C 90.000,E1 110.972} C_DIS
LIN {X 0.175,Y -578.319,Z 1061.411,A 0.000,B 0.000,C 90.000,E1 109.939} C_DIS
LIN {X -0.218,Y -573.939,Z 1061.409,A 0.000,B 0.000,C 90.000,E1 109.631} C_DIS
LIN {X 0.044,Y -569.461,Z 1061.407,A 0.000,B 0.000,C 90.000,E1 109.268} C_DIS
LIN {X -0.153,Y -561.078,Z 1061.404,A 0.000,B 0.000,C 90.000,E1 108.779} C_DIS
LIN {X -0.185,Y -554.492,Z 1061.402,A 0.000,B 0.000,C 90.000,E1 108.417} C_DIS
LIN {X 0.055,Y -549.407,Z 1061.400,A 0.000,B 0.000,C 90.000,E1 108.055} C_DIS
LIN {X -0.174,Y -547.684,Z 1061.399,A 0.000,B 0.000,C 90.000,E1 107.873} C_DIS
LIN {X -0.216,Y -547.662,Z 1061.399,A 0.000,B 0.000,C 90.000,E1 107.873} C_DIS
LIN {X 0.264,Y -547.308,Z 1061.397,A 0.000,B 0.000,C 90.000,E1 107.511} C_DIS
LIN {X 0.112,Y -548.648,Z 1061.384,A 0.000,B 0.000,C 90.000,E1 105.134} C_DIS
LIN {X -0.168,Y -550.685,Z 1061.369,A 0.000,B 0.000,C 90.000,E1 102.355} C_DIS
LIN {X 0.093,Y -552.518,Z 1061.358,A 0.000,B 0.000,C 90.000,E1 100.366} C_DIS
LIN {X 0.089,Y -554.338,Z 1061.348,A 0.000,B 0.000,C 90.000,E1 98.690} C_DIS
LIN {X 0.265,Y -556.602,Z 1061.338,A 0.000,B 0.000,C 90.000,E1 96.720} C_DIS
LIN {X 0.093,Y -557.815,Z 1061.331,A 0.000,B 0.000,C 90.000,E1 95.625} C_DIS
LIN {X -0.065,Y -558.856,Z 1061.325,A 0.000,B 0.000,C 90.000,E1 94.531} C_DIS
LIN {X -0.137,Y -559.816,Z 1061.318,A 0.000,B 0.000,C 90.000,E1 93.151} C_DIS
LIN {X -0.137,Y -560.600,Z 1061.308,A 0.000,B 0.000,C 90.000,E1 91.489} C_DIS
LIN {X -0.221,Y -561.183,Z 1061.301,A 0.000,B 0.000,C 90.000,E1 90.115} C_DIS
LIN {X -0.084,Y -561.846,Z 1061.290,A 0.000,B 0.000,C 90.000,E1 88.165} C_DIS
LIN {X 0.067,Y -562.564,Z 1061.279,A 0.000,B 0.000,C 90.000,E1 86.216} C_DIS
LIN {X 0.155,Y -563.179,Z 1061.270,A 0.000,B 0.000,C 90.000,E1 84.552} C_DIS
LIN {X -0.189,Y -563.566,Z 1061.261,A 0.000,B 0.000,C 90.000,E1 82.932} C_DIS
LIN {X 0.124,Y -564.157,Z 1061.250,A 0.000,B 0.000,C 90.000,E1 80.971} C_DIS
LIN {X -0.161,Y -565.108,Z 1061.236,A 0.000,B 0.000,C 90.000,E1 78.522} C_DIS
LIN {X 0.127,Y -565.825,Z 1061.229,A 0.000,B 0.000,C 90.000,E1 77.117} C_DIS
LIN {X 0.279,Y -567.281,Z 1061.215,A 0.000,B 0.000,C 90.000,E1 74.629} C_DIS
LIN {X -0.031,Y -568.544,Z 1061.206,A 0.000,B 0.000,C 90.000,E1 73.015} C_DIS
LIN {X -0.359,Y -570.301,Z 1061.193,A 0.000,B 0.000,C 90.000,E1 70.859} C_DIS
LIN {X 0.126,Y -571.475,Z 1061.186,A 0.000,B 0.000,C 90.000,E1 69.444} C_DIS
LIN {X 0.088,Y -573.012,Z 1061.175,A 0.000,B 0.000,C 90.000,E1 67.539} C_DIS
LIN {X -0.068,Y -574.134,Z 1061.166,A 0.000,B 0.000,C 90.000,E1 65.921} C_DIS
LIN {X -0.126,Y -575.310,Z 1061.156,A 0.000,B 0.000,C 90.000,E1 64.024} C_DIS
LIN {X 0.244,Y -576.201,Z 1061.147,A 0.000,B 0.000,C 90.000,E1 62.359} C_DIS
LIN {X 0.112,Y -577.045,Z 1061.138,A 0.000,B 0.000,C 90.000,E1 60.745} C_DIS
LIN {X -0.076,Y -577.666,Z 1061.130,A 0.000,B 0.000,C 90.000,E1 59.410} C_DIS
LIN {X -0.099,Y -578.310,Z 1061.121,A 0.000,B 0.000,C 90.000,E1 57.788} C_DIS
LIN {X -0.113,Y -579.016,Z 1061.112,A 0.000,B 0.000,C 90.000,E1 56.167} C_DIS
LIN {X -0.114,Y -579.544,Z 1061.102,A 0.000,B 0.000,C 90.000,E1 54.276} C_DIS
LIN {X -0.262,Y -579.732,Z 1061.095,A 0.000,B 0.000,C 90.000,E1 53.210} C_DIS
LIN {X 0.279,Y -579.727,Z 1061.087,A 0.000,B 0.000,C 90.000,E1 51.537} C_DIS
LIN {X 0.323,Y -579.528,Z 1061.082,A 0.000,B 0.000,C 90.000,E1 50.723} C_DIS
LIN {X -0.036,Y -578.847,Z 1061.073,A 0.000,B 0.000,C 90.000,E1 49.138} C_DIS
LIN {X -0.285,Y -578.345,Z 1061.067,A 0.000,B 0.000,C 90.000,E1 48.081} C_DIS
LIN {X -0.012,Y -577.475,Z 1061.059,A 0.000,B 0.000,C 90.000,E1 46.701} C_DIS
LIN {X -0.035,Y -576.823,Z 1061.055,A 0.000,B 0.000,C 90.000,E1 45.891} C_DIS
LIN {X -0.061,Y -575.994,Z 1061.050,A 0.000,B 0.000,C 90.000,E1 45.081} C_DIS
LIN {X -0.380,Y -574.708,Z 1061.044,A 0.000,B 0.000,C 90.000,E1 44.028} C_DIS
LIN {X -0.080,Y -572.330,Z 1061.035,A 0.000,B 0.000,C 90.000,E1 42.366} C_DIS
LIN {X 0.080,Y -569.973,Z 1061.028,A 0.000,B 0.000,C 90.000,E1 40.987} C_DIS
LIN {X -0.175,Y -566.959,Z 1061.020,A 0.000,B 0.000,C 90.000,E1 39.644} C_DIS
LIN {X -0.151,Y -564.030,Z 1061.014,A 0.000,B 0.000,C 90.000,E1 38.543} C_DIS
LIN {X 0.069,Y -562.449,Z 1061.011,A 0.000,B 0.000,C 90.000,E1 37.971} C_DIS
LIN {X -0.070,Y -559.788,Z 1061.006,A 0.000,B 0.000,C 90.000,E1 37.156} C_DIS
LIN {X 0.118,Y -557.867,Z 1061.003,A 0.000,B 0.000,C 90.000,E1 36.583} C_DIS
LIN {X 0.290,Y -555.753,Z 1061.000,A 0.000,B 0.000,C 90.000,E1 36.011} C_DIS
LIN {X -0.255,Y -552.196,Z 1060.996,A 0.000,B 0.000,C 90.000,E1 35.231} C_DIS
LIN {X 0.325,Y -549.701,Z 1060.993,A 0.000,B 0.000,C 90.000,E1 34.612} C_DIS
LIN {X 0.165,Y -545.786,Z 1060.988,A 0.000,B 0.000,C 90.000,E1 33.785} C_DIS
LIN {X -0.015,Y -539.968,Z 1060.982,A 0.000,B 0.000,C 90.000,E1 32.673} C_DIS
LIN {X 0.174,Y -535.206,Z 1060.977,A 0.000,B 0.000,C 90.000,E1 31.799} C_DIS
LIN {X 0.308,Y -530.098,Z 1060.972,A 0.000,B 0.000,C 90.000,E1 30.924} C_DIS
LIN {X -0.182,Y -525.389,Z 1060.968,A 0.000,B 0.000,C 90.000,E1 30.256} C_DIS
LIN {X -0.223,Y -520.299,Z 1060.964,A 0.000,B 0.000,C 90.000,E1 29.539} C_DIS
LIN {X -0.171,Y -515.997,Z 1060.961,A 0.000,B 0.000,C 90.000,E1 28.949} C_DIS
LIN {X -0.151,Y -511.331,Z 1060.958,A 0.000,B 0.000,C 90.000,E1 28.359} C_DIS
LIN {X 0.020,Y -507.685,Z 1060.955,A 0.000,B 0.000,C 90.000,E1 27.897} C_DIS
LIN {X -0.022,Y -502.536,Z 1060.952,A 0.000,B 0.000,C 90.000,E1 27.308} C_DIS
LIN {X -0.159,Y -497.113,Z 1060.948,A 0.000,B 0.000,C 90.000,E1 26.744} C_DIS
LIN {X -0.064,Y -490.318,Z 1060.945,A 0.000,B 0.000,C 90.000,E1 26.027} C_DIS
LIN {X -0.138,Y -480.574,Z 1060.939,A 0.000,B 0.000,C 90.000,E1 25.079} C_DIS
LIN {X -0.170,Y -471.857,Z 1060.935,A 0.000,B 0.000,C 90.000,E1 24.259} C_DIS
LIN {X -0.007,Y -465.821,Z 1060.932,A 0.000,B 0.000,C 90.000,E1 23.695} C_DIS
LIN {X 0.124,Y -455.163,Z 1060.927,A 0.000,B 0.000,C 90.000,E1 22.770} C_DIS
LIN {X -0.234,Y -445.998,Z 1060.922,A 0.000,B 0.000,C 90.000,E1 22.025} C_DIS
LIN {X -0.167,Y -426.763,Z 1060.912,A 0.000,B 0.000,C 90.000,E1 20.248} C_DIS
LIN {X -0.046,Y -414.010,Z 1060.905,A 0.000,B 0.000,C 90.000,E1 18.906} C_DIS
LIN {X -0.066,Y -401.664,Z 1060.897,A 0.000,B 0.000,C 90.000,E1 17.457} C_DIS
LIN {X 0.128,Y -399.130,Z 1060.895,A 0.000,B 0.000,C 90.000,E1 17.094} C_DIS
LIN {X 0.042,Y -395.273,Z 1060.892,A 0.000,B 0.000,C 90.000,E1 16.496} C_DIS
LIN {X 0.078,Y -394.347,Z 1060.891,A 0.000,B 0.000,C 90.000,E1 16.315} C_DIS
LIN {X -0.105,Y -392.787,Z 1060.889,A 0.000,B 0.000,C 90.000,E1 15.969} C_DIS
LIN {X -0.025,Y -391.800,Z 1060.886,A 0.000,B 0.000,C 90.000,E1 15.426} C_DIS
LIN {X -0.093,Y -391.610,Z 1060.883,A 0.000,B 0.000,C 90.000,E1 14.883} C_DIS
LIN {X -0.162,Y -392.345,Z 1060.877,A 0.000,B 0.000,C 90.000,E1 13.828} C_DIS
LIN {X 0.027,Y -398.494,Z 1060.853,A 0.000,B 0.000,C 90.000,E1 9.557} C_DIS
LIN {X -0.047,Y -400.942,Z 1060.845,A 0.000,B 0.000,C 90.000,E1 8.163} C_DIS
LIN {X 0.185,Y -407.509,Z 1060.828,A 0.000,B 0.000,C 90.000,E1 4.992} C_DIS
LIN {X 0.176,Y -410.055,Z 1060.822,A 0.000,B 0.000,C 90.000,E1 3.955} C_DIS
LIN {X 0.156,Y -411.654,Z 1060.819,A 0.000,B 0.000,C 90.000,E1 3.440} C_DIS
LIN {X 0.174,Y -413.620,Z 1060.817,A 0.000,B 0.000,C 90.000,E1 3.094} C_DIS
LIN {X 0.175,Y -415.855,Z 1060.815,A 0.000,B 0.000,C 90.000,E1 2.751} C_DIS
LIN {X 0.178,Y -417.157,Z 1060.815,A 0.000,B 0.000,C 90.000,E1 2.579} C_DIS
LIN {X 0.033,Y -422.438,Z 1060.812,A 0.000,B 0.000,C 90.000,E1 2.121} C_DIS
LIN {X 0.155,Y -431.133,Z 1060.809,A 0.000,B 0.000,C 90.000,E1 1.547} C_DIS
LIN {X 0.010,Y -451.014,Z 1060.802,A 0.000,B 0.000,C 90.000,E1 0.286} C_DIS
LIN {X -0.234,Y -467.235,Z 1060.796,A 0.000,B 0.000,C 90.000,E1 359.312} C_DIS
LIN {X 0.106,Y -485.283,Z 1060.790,A 0.000,B 0.000,C 90.000,E1 358.165} C_DIS
LIN {X 0.031,Y -498.000,Z 1060.785,A 0.000,B 0.000,C 90.000,E1 357.364} C_DIS
LIN {X -0.178,Y -504.307,Z 1060.783,A 0.000,B 0.000,C 90.000,E1 356.963} C_DIS
LIN {X -0.011,Y -510.507,Z 1060.781,A 0.000,B 0.000,C 90.000,E1 356.502} C_DIS
LIN {X 0.009,Y -517.957,Z 1060.777,A 0.000,B 0.000,C 90.000,E1 355.927} C_DIS
LIN {X -0.163,Y -523.775,Z 1060.775,A 0.000,B 0.000,C 90.000,E1 355.469} C_DIS
LIN {X 0.066,Y -529.441,Z 1060.772,A 0.000,B 0.000,C 90.000,E1 354.951} C_DIS
LIN {X -0.049,Y -536.158,Z 1060.768,A 0.000,B 0.000,C 90.000,E1 354.318} C_DIS
LIN {X -0.004,Y -542.533,Z 1060.765,A 0.000,B 0.000,C 90.000,E1 353.628} C_DIS
LIN {X 0.150,Y -547.422,Z 1060.762,A 0.000,B 0.000,C 90.000,E1 353.053} C_DIS
LIN {X 0.096,Y -552.743,Z 1060.758,A 0.000,B 0.000,C 90.000,E1 352.356} C_DIS
LIN {X 0.254,Y -556.694,Z 1060.755,A 0.000,B 0.000,C 90.000,E1 351.781} C_DIS
LIN {X 0.274,Y -561.052,Z 1060.751,A 0.000,B 0.000,C 90.000,E1 351.084} C_DIS
LIN {X 0.022,Y -564.339,Z 1060.748,A 0.000,B 0.000,C 90.000,E1 350.557} C_DIS
LIN {X 0.113,Y -568.004,Z 1060.744,A 0.000,B 0.000,C 90.000,E1 349.859} C_DIS
LIN {X -0.191,Y -570.732,Z 1060.741,A 0.000,B 0.000,C 90.000,E1 349.342} C_DIS
LIN {X 0.262,Y -575.158,Z 1060.735,A 0.000,B 0.000,C 90.000,E1 348.342} C_DIS
LIN {X -0.259,Y -580.374,Z 1060.729,A 0.000,B 0.000,C 90.000,E1 347.173} C_DIS
LIN {X 0.082,Y -584.625,Z 1060.723,A 0.000,B 0.000,C 90.000,E1 346.061} C_DIS
LIN {X 0.056,Y -588.641,Z 1060.717,A 0.000,B 0.000,C 90.000,E1 344.991} C_DIS
LIN {X 0.088,Y -592.546,Z 1060.711,A 0.000,B 0.000,C 90.000,E1 343.921} C_DIS
LIN {X 0.049,Y -597.218,Z 1060.703,A 0.000,B 0.000,C 90.000,E1 342.598} C_DIS
LIN {X 0.091,Y -601.460,Z 1060.696,A 0.000,B 0.000,C 90.000,E1 341.275} C_DIS
LIN {X -0.375,Y -605.244,Z 1060.689,A 0.000,B 0.000,C 90.000,E1 340.007} C_DIS
LIN {X 0.210,Y -608.690,Z 1060.682,A 0.000,B 0.000,C 90.000,E1 338.646} C_DIS
LIN {X -0.172,Y -610.650,Z 1060.677,A 0.000,B 0.000,C 90.000,E1 337.901} C_DIS
LIN {X -0.285,Y -613.578,Z 1060.670,A 0.000,B 0.000,C 90.000,E1 336.613} C_DIS
LIN {X 0.159,Y -615.589,Z 1060.664,A 0.000,B 0.000,C 90.000,E1 335.537} C_DIS
LIN {X -0.184,Y -617.353,Z 1060.658,A 0.000,B 0.000,C 90.000,E1 334.537} C_DIS
LIN {X -0.230,Y -618.489,Z 1060.654,A 0.000,B 0.000,C 90.000,E1 333.768} C_DIS
LIN {X -0.272,Y -619.929,Z 1060.648,A 0.000,B 0.000,C 90.000,E1 332.743} C_DIS
LIN {X -0.008,Y -621.456,Z 1060.641,A 0.000,B 0.000,C 90.000,E1 331.435} C_DIS
LIN {X -0.018,Y -622.297,Z 1060.637,A 0.000,B 0.000,C 90.000,E1 330.667} C_DIS
LIN {X -0.257,Y -623.151,Z 1060.631,A 0.000,B 0.000,C 90.000,E1 329.665} C_DIS
LIN {X 0.371,Y -623.791,Z 1060.624,A 0.000,B 0.000,C 90.000,E1 328.329} C_DIS
LIN {X 0.158,Y -624.133,Z 1060.620,A 0.000,B 0.000,C 90.000,E1 327.582} C_DIS
LIN {X -0.064,Y -624.202,Z 1060.614,A 0.000,B 0.000,C 90.000,E1 326.580} C_DIS
LIN {X 0.051,Y -624.085,Z 1060.609,A 0.000,B 0.000,C 90.000,E1 325.548} C_DIS
LIN {X -0.014,Y -623.809,Z 1060.602,A 0.000,B 0.000,C 90.000,E1 324.276} C_DIS
LIN {X 0.422,Y -623.047,Z 1060.590,A 0.000,B 0.000,C 90.000,E1 322.190} C_DIS
LIN {X -0.189,Y -622.201,Z 1060.573,A 0.000,B 0.000,C 90.000,E1 319.175} C_DIS
LIN {X -0.310,Y -621.942,Z 1060.568,A 0.000,B 0.000,C 90.000,E1 318.162} C_DIS
LIN {X 0.021,Y -621.356,Z 1060.557,A 0.000,B 0.000,C 90.000,E1 316.338} C_DIS
LIN {X -0.107,Y -621.082,Z 1060.552,A 0.000,B 0.000,C 90.000,E1 315.324} C_DIS
LIN {X 0.060,Y -620.641,Z 1060.540,A 0.000,B 0.000,C 90.000,E1 313.257} C_DIS
LIN {X -0.374,Y -620.109,Z 1060.532,A 0.000,B 0.000,C 90.000,E1 311.757} C_DIS
LIN {X -0.212,Y -619.445,Z 1060.525,A 0.000,B 0.000,C 90.000,E1 310.458} C_DIS
LIN {X 0.102,Y -619.420,Z 1060.523,A 0.000,B 0.000,C 90.000,E1 310.172} C_DIS
LIN {X 0.002,Y -618.629,Z 1060.513,A 0.000,B 0.000,C 90.000,E1 308.382} C_DIS
LIN {X -0.016,Y -618.219,Z 1060.503,A 0.000,B 0.000,C 90.000,E1 306.583} C_DIS
LIN {X 0.377,Y -618.092,Z 1060.498,A 0.000,B 0.000,C 90.000,E1 305.518} C_DIS
LIN {X 0.140,Y -617.838,Z 1060.495,A 0.000,B 0.000,C 90.000,E1 305.025} C_DIS
LIN {X 0.099,Y -618.004,Z 1060.493,A 0.000,B 0.000,C 90.000,E1 304.771} C_DIS
LIN {X -0.065,Y -617.995,Z 1060.486,A 0.000,B 0.000,C 90.000,E1 303.499} C_DIS
LIN {X 0.212,Y -617.769,Z 1060.483,A 0.000,B 0.000,C 90.000,E1 302.959} C_DIS
LIN {X -0.337,Y -617.975,Z 1060.482,A 0.000,B 0.000,C 90.000,E1 302.752} C_DIS
LIN {X -0.332,Y -618.003,Z 1060.475,A 0.000,B 0.000,C 90.000,E1 301.465} C_DIS
LIN {X -0.055,Y -617.781,Z 1060.472,A 0.000,B 0.000,C 90.000,E1 300.924} C_DIS
LIN {X -0.076,Y -617.925,Z 1060.470,A 0.000,B 0.000,C 90.000,E1 300.669} C_DIS
LIN {X -0.389,Y -618.091,Z 1060.463,A 0.000,B 0.000,C 90.000,E1 299.411} C_DIS
LIN {X -0.162,Y -617.971,Z 1060.456,A 0.000,B 0.000,C 90.000,E1 298.103} C_DIS
LIN {X 0.054,Y -617.324,Z 1060.449,A 0.000,B 0.000,C 90.000,E1 296.796} C_DIS
LIN {X -0.296,Y -616.139,Z 1060.442,A 0.000,B 0.000,C 90.000,E1 295.540} C_DIS
LIN {X 0.182,Y -614.546,Z 1060.436,A 0.000,B 0.000,C 90.000,E1 294.463} C_DIS
LIN {X 0.101,Y -612.950,Z 1060.432,A 0.000,B 0.000,C 90.000,E1 293.695} C_DIS
LIN {X -0.208,Y -611.606,Z 1060.429,A 0.000,B 0.000,C 90.000,E1 293.206} C_DIS
LIN {X -0.244,Y -610.771,Z 1060.427,A 0.000,B 0.000,C 90.000,E1 292.950} C_DIS
LIN {X 0.002,Y -608.826,Z 1060.425,A 0.000,B 0.000,C 90.000,E1 292.408} C_DIS
LIN {X -0.096,Y -606.470,Z 1060.422,A 0.000,B 0.000,C 90.000,E1 291.897} C_DIS
LIN {X 0.155,Y -604.091,Z 1060.419,A 0.000,B 0.000,C 90.000,E1 291.482} C_DIS
LIN {X 0.013,Y -600.102,Z 1060.417,A 0.000,B 0.000,C 90.000,E1 290.972} C_DIS
LIN {X -0.062,Y -595.055,Z 1060.414,A 0.000,B 0.000,C 90.000,E1 290.482} C_DIS
LIN {X 0.088,Y -590.960,Z 1060.412,A 0.000,B 0.000,C 90.000,E1 290.120} C_DIS
LIN {X 0.190,Y -589.432,Z 1060.411,A 0.000,B 0.000,C 90.000,E1 289.993} C_DIS
LIN {X 0.091,Y -587.395,Z 1060.411,A 0.000,B 0.000,C 90.000,E1 289.885} C_DIS
LIN {X -0.108,Y -583.506,Z 1060.409,A 0.000,B 0.000,C 90.000,E1 289.631} C_DIS
LIN {X -0.321,Y -578.002,Z 1060.408,A 0.000,B 0.000,C 90.000,E1 289.396} C_DIS
LIN {X -0.256,Y -576.087,Z 1060.407,A 0.000,B 0.000,C 90.000,E1 289.268} C_DIS
LIN {X 0.039,Y -574.114,Z 1060.406,A 0.000,B 0.000,C 90.000,E1 289.141} C_DIS
LIN {X -0.134,Y -566.915,Z 1060.405,A 0.000,B 0.000,C 90.000,E1 288.852} C_DIS
LIN {X -0.132,Y -564.116,Z 1060.404,A 0.000,B 0.000,C 90.000,E1 288.779} C_DIS
LIN {X -0.253,Y -557.898,Z 1060.404,A 0.000,B 0.000,C 90.000,E1 288.725} C_DIS
LIN {X -0.286,Y -551.484,Z 1060.404,A 0.000,B 0.000,C 90.000,E1 288.725} C_DIS
LIN {X -0.079,Y -546.871,Z 1060.404,A 0.000,B 0.000,C 90.000,E1 288.652} C_DIS
LIN {X -0.134,Y -546.355,Z 1060.404,A 0.000,B 0.000,C 90.000,E1 288.652} C_DIS
LIN {X -0.171,Y -546.113,Z 1060.402,A 0.000,B 0.000,C 90.000,E1 288.362} C_DIS
LIN {X 0.076,Y -545.614,Z 1060.400,A 0.000,B 0.000,C 90.000,E1 288.055} C_DIS
LIN {X -0.078,Y -545.372,Z 1060.400,A 0.000,B 0.000,C 90.000,E1 288.000} C_DIS
LIN {X -0.154,Y -544.559,Z 1060.386,A 0.000,B 0.000,C 90.000,E1 285.536} C_DIS
LIN {X -0.207,Y -544.290,Z 1060.380,A 0.000,B 0.000,C 90.000,E1 284.411} C_DIS
LIN {X 0.138,Y -543.921,Z 1060.374,A 0.000,B 0.000,C 90.000,E1 283.244} C_DIS
LIN {X 0.244,Y -543.010,Z 1060.364,A 0.000,B 0.000,C 90.000,E1 281.535} C_DIS
LIN {X 0.189,Y -541.841,Z 1060.353,A 0.000,B 0.000,C 90.000,E1 279.557} C_DIS
LIN {X -0.045,Y -541.020,Z 1060.345,A 0.000,B 0.000,C 90.000,E1 278.163} C_DIS
LIN {X 0.229,Y -540.005,Z 1060.336,A 0.000,B 0.000,C 90.000,E1 276.429} C_DIS
LIN {X -0.121,Y -538.998,Z 1060.326,A 0.000,B 0.000,C 90.000,E1 274.759} C_DIS
LIN {X -0.001,Y -538.075,Z 1060.317,A 0.000,B 0.000,C 90.000,E1 273.037} C_DIS
LIN {X 0.072,Y -537.127,Z 1060.307,A 0.000,B 0.000,C 90.000,E1 271.318} C_DIS
LIN {X 0.119,Y -536.105,Z 1060.298,A 0.000,B 0.000,C 90.000,E1 269.599} C_DIS
LIN {X 0.155,Y -535.085,Z 1060.288,A 0.000,B 0.000,C 90.000,E1 267.879} C_DIS
LIN {X 0.166,Y -533.994,Z 1060.279,A 0.000,B 0.000,C 90.000,E1 266.159} C_DIS
LIN {X 0.190,Y -532.989,Z 1060.271,A 0.000,B 0.000,C 90.000,E1 264.723} C_DIS
LIN {X 0.215,Y -532.065,Z 1060.264,A 0.000,B 0.000,C 90.000,E1 263.571} C_DIS
LIN {X -0.236,Y -531.000,Z 1060.258,A 0.000,B 0.000,C 90.000,E1 262.470} C_DIS
LIN {X -0.086,Y -528.228,Z 1060.244,A 0.000,B 0.000,C 90.000,E1 259.859} C_DIS
LIN {X -0.023,Y -526.335,Z 1060.234,A 0.000,B 0.000,C 90.000,E1 258.117} C_DIS
LIN {X 0.190,Y -524.746,Z 1060.226,A 0.000,B 0.000,C 90.000,E1 256.645} C_DIS
LIN {X -0.130,Y -523.254,Z 1060.218,A 0.000,B 0.000,C 90.000,E1 255.227} C_DIS
LIN {X 0.157,Y -521.444,Z 1060.208,A 0.000,B 0.000,C 90.000,E1 253.449} C_DIS
LIN {X 0.065,Y -519.929,Z 1060.200,A 0.000,B 0.000,C 90.000,E1 252.000} C_DIS
LIN {X -0.051,Y -518.288,Z 1060.192,A 0.000,B 0.000,C 90.000,E1 250.550} C_DIS
LIN {X 0.111,Y -516.167,Z 1060.182,A 0.000,B 0.000,C 90.000,E1 248.773} C_DIS
LIN {X 0.093,Y -514.180,Z 1060.174,A 0.000,B 0.000,C 90.000,E1 247.305} C_DIS
LIN {X 0.107,Y -512.533,Z 1060.167,A 0.000,B 0.000,C 90.000,E1 246.125} C_DIS
LIN {X -0.050,Y -510.303,Z 1060.159,A 0.000,B 0.000,C 90.000,E1 244.665} C_DIS
LIN {X -0.015,Y -507.888,Z 1060.151,A 0.000,B 0.000,C 90.000,E1 243.179} C_DIS
LIN {X 0.033,Y -506.467,Z 1060.146,A 0.000,B 0.000,C 90.000,E1 242.281} C_DIS
LIN {X -0.131,Y -503.434,Z 1060.136,A 0.000,B 0.000,C 90.000,E1 240.511} C_DIS
LIN {X 0.021,Y -500.647,Z 1060.128,A 0.000,B 0.000,C 90.000,E1 238.997} C_DIS
LIN {X -0.050,Y -497.907,Z 1060.120,A 0.000,B 0.000,C 90.000,E1 237.502} C_DIS
LIN {X -0.033,Y -495.639,Z 1060.113,A 0.000,B 0.000,C 90.000,E1 236.294} C_DIS
LIN {X -0.080,Y -492.085,Z 1060.103,A 0.000,B 0.000,C 90.000,E1 234.482} C_DIS
LIN {X 0.001,Y -489.379,Z 1060.096,A 0.000,B 0.000,C 90.000,E1 233.256} C_DIS
LIN {X 0.219,Y -484.491,Z 1060.084,A 0.000,B 0.000,C 90.000,E1 231.090} C_DIS
LIN {X 0.226,Y -479.645,Z 1060.072,A 0.000,B 0.000,C 90.000,E1 228.933} C_DIS
LIN {X 0.161,Y -476.431,Z 1060.063,A 0.000,B 0.000,C 90.000,E1 227.391} C_DIS
LIN {X -0.211,Y -472.721,Z 1060.053,A 0.000,B 0.000,C 90.000,E1 225.567} C_DIS
LIN {X 0.161,Y -470.336,Z 1060.046,A 0.000,B 0.000,C 90.000,E1 224.271} C_DIS
LIN {X -0.001,Y -466.672,Z 1060.036,A 0.000,B 0.000,C 90.000,E1 222.405} C_DIS
LIN {X -0.246,Y -462.810,Z 1060.025,A 0.000,B 0.000,C 90.000,E1 220.539} C_DIS
LIN {X 0.107,Y -458.857,Z 1060.015,A 0.000,B 0.000,C 90.000,E1 218.588} C_DIS
LIN {X 0.155,Y -455.015,Z 1060.004,A 0.000,B 0.000,C 90.000,E1 216.664} C_DIS
LIN {X -0.228,Y -451.664,Z 1059.995,A 0.000,B 0.000,C 90.000,E1 215.105} C_DIS
LIN {X 0.068,Y -448.227,Z 1059.986,A 0.000,B 0.000,C 90.000,E1 213.452} C_DIS
LIN {X 0.290,Y -444.945,Z 1059.977,A 0.000,B 0.000,C 90.000,E1 211.799} C_DIS
LIN {X 0.028,Y -440.896,Z 1059.966,A 0.000,B 0.000,C 90.000,E1 209.873} C_DIS
LIN {X 0.022,Y -437.435,Z 1059.957,A 0.000,B 0.000,C 90.000,E1 208.231} C_DIS
LIN {X 0.131,Y -434.150,Z 1059.948,A 0.000,B 0.000,C 90.000,E1 206.565} C_DIS
LIN {X 0.175,Y -430.848,Z 1059.938,A 0.000,B 0.000,C 90.000,E1 204.899} C_DIS
LIN {X -0.084,Y -424.884,Z 1059.920,A 0.000,B 0.000,C 90.000,E1 201.589} C_DIS
LIN {X -0.157,Y -421.897,Z 1059.909,A 0.000,B 0.000,C 90.000,E1 199.577} C_DIS
LIN {X 0.101,Y -420.001,Z 1059.897,A 0.000,B 0.000,C 90.000,E1 197.511} C_DIS
LIN {X -0.086,Y -419.634,Z 1059.894,A 0.000,B 0.000,C 90.000,E1 196.858} C_DIS
LIN {X 0.131,Y -419.558,Z 1059.890,A 0.000,B 0.000,C 90.000,E1 196.150} C_DIS
LIN {X 0.059,Y -419.827,Z 1059.886,A 0.000,B 0.000,C 90.000,E1 195.481} C_DIS
LIN {X -0.071,Y -420.841,Z 1059.880,A 0.000,B 0.000,C 90.000,E1 194.481} C_DIS
LIN {X 0.159,Y -422.186,Z 1059.877,A 0.000,B 0.000,C 90.000,E1 193.772} C_DIS
LIN {X -0.012,Y -424.114,Z 1059.873,A 0.000,B 0.000,C 90.000,E1 193.119} C_DIS
LIN {X -0.084,Y -428.172,Z 1059.867,A 0.000,B 0.000,C 90.000,E1 192.119} C_DIS
LIN {X -0.075,Y -433.274,Z 1059.862,A 0.000,B 0.000,C 90.000,E1 191.130} C_DIS
LIN {X 0.142,Y -442.014,Z 1059.854,A 0.000,B 0.000,C 90.000,E1 189.613} C_DIS
LIN {X 0.200,Y -453.366,Z 1059.844,A 0.000,B 0.000,C 90.000,E1 187.814} C_DIS
LIN {X -0.036,Y -460.592,Z 1059.837,A 0.000,B 0.000,C 90.000,E1 186.720} C_DIS
LIN {X 0.184,Y -466.687,Z 1059.832,A 0.000,B 0.000,C 90.000,E1 185.739} C_DIS
LIN {X -0.155,Y -471.585,Z 1059.828,A 0.000,B 0.000,C 90.000,E1 184.992} C_DIS
LIN {X 0.026,Y -476.312,Z 1059.823,A 0.000,B 0.000,C 90.000,E1 184.188} C_DIS
LIN {X 0.232,Y -483.683,Z 1059.816,A 0.000,B 0.000,C 90.000,E1 182.922} C_DIS
LIN {X 0.033,Y -490.920,Z 1059.810,A 0.000,B 0.000,C 90.000,E1 181.718} C_DIS
LIN {X -0.208,Y -499.692,Z 1059.801,A 0.000,B 0.000,C 90.000,E1 180.229} C_DIS
LIN {X 0.015,Y -507.188,Z 1059.794,A 0.000,B 0.000,C 90.000,E1 178.854} C_DIS
LIN {X -0.129,Y -514.607,Z 1059.786,A 0.000,B 0.000,C 90.000,E1 177.535} C_DIS
LIN {X -0.174,Y -523.439,Z 1059.777,A 0.000,B 0.000,C 90.000,E1 175.927} C_DIS
LIN {X -0.038,Y -532.128,Z 1059.768,A 0.000,B 0.000,C 90.000,E1 174.318} C_DIS
LIN {X -0.215,Y -540.573,Z 1059.760,A 0.000,B 0.000,C 90.000,E1 172.761} C_DIS
LIN {X -0.249,Y -547.408,Z 1059.753,A 0.000,B 0.000,C 90.000,E1 171.489} C_DIS
LIN {X 0.200,Y -554.853,Z 1059.745,A 0.000,B 0.000,C 90.000,E1 170.038} C_DIS
LIN {X -0.063,Y -561.345,Z 1059.738,A 0.000,B 0.000,C 90.000,E1 168.814} C_DIS
LIN {X -0.230,Y -567.548,Z 1059.731,A 0.000,B 0.000,C 90.000,E1 167.589} C_DIS
LIN {X 0.068,Y -572.946,Z 1059.725,A 0.000,B 0.000,C 90.000,E1 166.464} C_DIS
LIN {X -0.206,Y -576.163,Z 1059.721,A 0.000,B 0.000,C 90.000,E1 165.811} C_DIS
LIN {X -0.109,Y -582.369,Z 1059.714,A 0.000,B 0.000,C 90.000,E1 164.448} C_DIS
LIN {X -0.157,Y -587.041,Z 1059.708,A 0.000,B 0.000,C 90.000,E1 163.378} C_DIS
LIN {X -0.150,Y -591.531,Z 1059.702,A 0.000,B 0.000,C 90.000,E1 162.308} C_DIS
LIN {X 0.094,Y -595.672,Z 1059.696,A 0.000,B 0.000,C 90.000,E1 161.221} C_DIS
LIN {X -0.167,Y -599.587,Z 1059.690,A 0.000,B 0.000,C 90.000,E1 160.188} C_DIS
LIN {X -0.165,Y -603.312,Z 1059.684,A 0.000,B 0.000,C 90.000,E1 159.135} C_DIS
LIN {X -0.327,Y -606.770,Z 1059.678,A 0.000,B 0.000,C 90.000,E1 158.103} C_DIS
LIN {X 0.063,Y -609.274,Z 1059.674,A 0.000,B 0.000,C 90.000,E1 157.283} C_DIS
LIN {X 0.208,Y -612.375,Z 1059.668,A 0.000,B 0.000,C 90.000,E1 156.230} C_DIS
LIN {X -0.173,Y -615.344,Z 1059.662,A 0.000,B 0.000,C 90.000,E1 155.229} C_DIS
LIN {X 0.274,Y -619.532,Z 1059.654,A 0.000,B 0.000,C 90.000,E1 153.640} C_DIS
LIN {X 0.249,Y -622.780,Z 1059.647,A 0.000,B 0.000,C 90.000,E1 152.359} C_DIS
LIN {X 0.042,Y -627.110,Z 1059.637,A 0.000,B 0.000,C 90.000,E1 150.589} C_DIS
LIN {X -0.091,Y -630.707,Z 1059.628,A 0.000,B 0.000,C 90.000,E1 149.076} C_DIS
LIN {X 0.163,Y -634.056,Z 1059.620,A 0.000,B 0.000,C 90.000,E1 147.533} C_DIS
LIN {X -0.084,Y -636.768,Z 1059.613,A 0.000,B 0.000,C 90.000,E1 146.294} C_DIS
LIN {X 0.105,Y -640.002,Z 1059.604,A 0.000,B 0.000,C 90.000,E1 144.769} C_DIS
LIN {X -0.194,Y -642.618,Z 1059.597,A 0.000,B 0.000,C 90.000,E1 143.543} C_DIS
LIN {X -0.023,Y -645.852,Z 1059.589,A 0.000,B 0.000,C 90.000,E1 142.029} C_DIS
LIN {X 0.202,Y -648.950,Z 1059.581,A 0.000,B 0.000,C 90.000,E1 140.517} C_DIS
LIN {X 0.341,Y -652.672,Z 1059.571,A 0.000,B 0.000,C 90.000,E1 138.771} C_DIS
LIN {X 0.082,Y -656.448,Z 1059.562,A 0.000,B 0.000,C 90.000,E1 137.067} C_DIS
LIN {X 0.339,Y -660.997,Z 1059.551,A 0.000,B 0.000,C 90.000,E1 135.081} C_DIS
LIN {X -0.218,Y -666.131,Z 1059.540,A 0.000,B 0.000,C 90.000,E1 133.176} C_DIS
LIN {X 0.272,Y -669.398,Z 1059.533,A 0.000,B 0.000,C 90.000,E1 131.919} C_DIS
LIN {X -0.047,Y -673.879,Z 1059.524,A 0.000,B 0.000,C 90.000,E1 130.253} C_DIS
LIN {X -0.296,Y -677.683,Z 1059.516,A 0.000,B 0.000,C 90.000,E1 128.830} C_DIS
LIN {X 0.048,Y -681.405,Z 1059.508,A 0.000,B 0.000,C 90.000,E1 127.363} C_DIS
LIN {X 0.046,Y -685.063,Z 1059.500,A 0.000,B 0.000,C 90.000,E1 125.931} C_DIS
LIN {X 0.081,Y -688.030,Z 1059.493,A 0.000,B 0.000,C 90.000,E1 124.739} C_DIS
LIN {X 0.372,Y -691.516,Z 1059.485,A 0.000,B 0.000,C 90.000,E1 123.293} C_DIS
LIN {X 0.126,Y -694.367,Z 1059.479,A 0.000,B 0.000,C 90.000,E1 122.133} C_DIS
LIN {X 0.163,Y -697.588,Z 1059.471,A 0.000,B 0.000,C 90.000,E1 120.718} C_DIS
LIN {X 0.328,Y -699.029,Z 1059.467,A 0.000,B 0.000,C 90.000,E1 120.001} C_DIS
LIN {X -0.099,Y -700.245,Z 1059.463,A 0.000,B 0.000,C 90.000,E1 119.333} C_DIS
LIN {X 0.095,Y -701.104,Z 1059.459,A 0.000,B 0.000,C 90.000,E1 118.615} C_DIS
LIN {X 0.050,Y -703.413,Z 1059.446,A 0.000,B 0.000,C 90.000,E1 116.283} C_DIS
LIN {X 0.241,Y -704.256,Z 1059.441,A 0.000,B 0.000,C 90.000,E1 115.335} C_DIS
LIN {X 0.160,Y -704.615,Z 1059.437,A 0.000,B 0.000,C 90.000,E1 114.643} C_DIS
LIN {X -0.202,Y -704.346,Z 1059.434,A 0.000,B 0.000,C 90.000,E1 114.207} C_DIS
LIN {X 0.082,Y -704.034,Z 1059.433,A 0.000,B 0.000,C 90.000,E1 113.951} C_DIS
LIN {X -0.281,Y -702.724,Z 1059.431,A 0.000,B 0.000,C 90.000,E1 113.515} C_DIS
LIN {X -0.003,Y -701.628,Z 1059.429,A 0.000,B 0.000,C 90.000,E1 113.259} C_DIS
LIN {X 0.263,Y -698.311,Z 1059.427,A 0.000,B 0.000,C 90.000,E1 112.770} C_DIS
LIN {X 0.393,Y -697.180,Z 1059.426,A 0.000,B 0.000,C 90.000,E1 112.642} C_DIS
LIN {X -0.387,Y -695.443,Z 1059.425,A 0.000,B 0.000,C 90.000,E1 112.589} C_DIS
LIN {X 0.116,Y -688.076,Z 1059.423,A 0.000,B 0.000,C 90.000,E1 112.206} C_DIS
LIN {X 0.307,Y -684.762,Z 1059.423,A 0.000,B 0.000,C 90.000,E1 112.078} C_DIS
LIN {X 0.194,Y -675.912,Z 1059.422,A 0.000,B 0.000,C 90.000,E1 111.972} C_DIS
LIN {X 0.128,Y -609.034,Z 1059.422,A 0.000,B 0.000,C 90.000,E1 111.972} C_DIS
LIN {X 0.005,Y -605.119,Z 1059.421,A 0.000,B 0.000,C 90.000,E1 111.844} C_DIS
LIN {X -0.216,Y -602.834,Z 1059.421,A 0.000,B 0.000,C 90.000,E1 111.770} C_DIS
LIN {X 0.269,Y -597.052,Z 1059.419,A 0.000,B 0.000,C 90.000,E1 111.408} C_DIS
LIN {X 0.192,Y -592.592,Z 1059.417,A 0.000,B 0.000,C 90.000,E1 111.099} C_DIS
LIN {X 0.203,Y -577.779,Z 1059.411,A 0.000,B 0.000,C 90.000,E1 109.885} C_DIS
LIN {X -0.187,Y -573.342,Z 1059.409,A 0.000,B 0.000,C 90.000,E1 109.577} C_DIS
LIN {X 0.146,Y -568.918,Z 1059.407,A 0.000,B 0.000,C 90.000,E1 109.214} C_DIS
LIN {X 0.145,Y -560.651,Z 1059.404,A 0.000,B 0.000,C 90.000,E1 108.725} C_DIS
LIN {X 0.109,Y -554.156,Z 1059.402,A 0.000,B 0.000,C 90.000,E1 108.362} C_DIS
LIN {X -0.213,Y -549.123,Z 1059.400,A 0.000,B 0.000,C 90.000,E1 108.055} C_DIS
LIN {X 0.245,Y -547.650,Z 1059.399,A 0.000,B 0.000,C 90.000,E1 107.819} C_DIS
LIN {X 0.213,Y -547.635,Z 1059.399,A 0.000,B 0.000,C 90.000,E1 107.819} C_DIS
LIN {X -0.092,Y -547.344,Z 1059.398,A 0.000,B 0.000,C 90.000,E1 107.638} C_DIS
LIN {X -0.050,Y -547.452,Z 1059.395,A 0.000,B 0.000,C 90.000,E1 107.040} C_DIS
LIN {X -0.242,Y -548.521,Z 1059.385,A 0.000,B 0.000,C 90.000,E1 105.371} C_DIS
LIN {X -0.100,Y -550.263,Z 1059.371,A 0.000,B 0.000,C 90.000,E1 102.827} C_DIS
LIN {X 0.156,Y -552.001,Z 1059.360,A 0.000,B 0.000,C 90.000,E1 100.838} C_DIS
LIN {X -0.191,Y -554.101,Z 1059.349,A 0.000,B 0.000,C 90.000,E1 98.916} C_DIS
LIN {X -0.280,Y -555.629,Z 1059.342,A 0.000,B 0.000,C 90.000,E1 97.530} C_DIS
LIN {X 0.151,Y -557.005,Z 1059.336,A 0.000,B 0.000,C 90.000,E1 96.372} C_DIS
LIN {X -0.019,Y -558.137,Z 1059.329,A 0.000,B 0.000,C 90.000,E1 95.277} C_DIS
LIN {X 0.256,Y -558.875,Z 1059.325,A 0.000,B 0.000,C 90.000,E1 94.416} C_DIS
LIN {X 0.187,Y -559.832,Z 1059.317,A 0.000,B 0.000,C 90.000,E1 93.037} C_DIS
LIN {X 0.098,Y -560.470,Z 1059.309,A 0.000,B 0.000,C 90.000,E1 91.661} C_DIS
